LIN {X 0,Y 513.004,Z 916.305,A -85,B 0,C 180,E1 22393.038,E2 22393.038} C_VEL
LIN {X 0,Y 508.896,Z 933.803,A -85,B 0,C 180,E1 22391.855,E2 22391.855} C_VEL
LIN {X 0,Y 504.363,Z 951.797,A -85,B 0,C 180,E1 22390.486,E2 22390.486} C_VEL
LIN {X 0,Y 498.956,Z 972.158,A -85,B 0,C 180,E1 22388.725,E2 22388.725} C_VEL
LIN {X 0,Y 493.08,Z 992.756,A -85,B 0,C 180,E1 22386.651,E2 22386.651} C_VEL
LIN {X 0,Y 488.236,Z 1008.925,A -85,B 0,C 180,E1 22384.788,E2 22384.788} C_VEL
LIN {X 0,Y 483.886,Z 1023.135,A -85,B 0,C 180,E1 22382.95,E2 22382.95} C_VEL
LIN {X 0,Y 479.724,Z 1036.506,A -85,B 0,C 180,E1 22381.021,E2 22381.021} C_VEL
LIN {X 0,Y 475.565,Z 1049.952,A -85,B 0,C 180,E1 22378.841,E2 22378.841} C_VEL
LIN {X 0,Y 470.95,Z 1065.021,A -85,B 0,C 180,E1 22376.057,E2 22376.057} C_VEL
LIN {X 0,Y 466.983,Z 1078.097,A -85,B 0,C 180,E1 22373.207,E2 22373.207} C_VEL
LIN {X 0,Y 464.273,Z 1087.644,A -85,B 0,C 180,E1 22370.835,E2 22370.835} C_VEL
LIN {X 0,Y 461.919,Z 1096.543,A -85,B 0,C 180,E1 22368.315,E2 22368.315} C_VEL
LIN {X 0,Y 459.756,Z 1105.63,A -85,B 0,C 180,E1 22365.33,E2 22365.33} C_VEL
LIN {X 0,Y 457.961,Z 1114.229,A -85,B 0,C 180,E1 22361.883,E2 22361.883} C_VEL
LIN {X 0,Y 456.92,Z 1120.716,A -85,B 0,C 180,E1 22358.628,E2 22358.628} C_VEL
LIN {X 0,Y 456.305,Z 1125.981,A -85,B 0,C 180,E1 22355.181,E2 22355.181} C_VEL
LIN {X 0,Y 456.039,Z 1129.45,A -85,B 0,C 180,E1 22351.898,E2 22351.898} C_VEL
LIN {X 0,Y 455.95,Z 1131.611,A -85,B 0,C 180,E1 22348.696,E2 22348.696} C_VEL
LIN {X 0,Y 455.919,Z 1132.456,A -85,B 0,C 180,E1 22345.371,E2 22345.371} C_VEL
LIN {X 0,Y 455.939,Z 1131.95,A -85,B 0,C 180,E1 22342.025,E2 22342.025} C_VEL
LIN {X 0,Y 456.017,Z 1130.259,A -85,B 0,C 180,E1 22338.803,E2 22338.803} C_VEL
LIN {X 0,Y 456.242,Z 1127.297,A -85,B 0,C 180,E1 22335.638,E2 22335.638} C_VEL
LIN {X 0,Y 456.832,Z 1122.324,A -85,B 0,C 180,E1 22331.943,E2 22331.943} C_VEL
LIN {X 0,Y 457.747,Z 1116.901,A -85,B 0,C 180,E1 22328.922,E2 22328.922} C_VEL
LIN {X 0,Y 459.142,Z 1110.45,A -85,B 0,C 180,E1 22326,E2 22326} C_VEL
LIN {X 0,Y 461.433,Z 1101.534,A -85,B 0,C 180,E1 22322.646,E2 22322.646} C_VEL
LIN {X 0,Y 464.2,Z 1091.739,A -85,B 0,C 180,E1 22319.63,E2 22319.63} C_VEL
LIN {X 0,Y 467.056,Z 1082.545,A -85,B 0,C 180,E1 22317.178,E2 22317.178} C_VEL
LIN {X 0,Y 470.587,Z 1071.658,A -85,B 0,C 180,E1 22314.636,E2 22314.636} C_VEL
LIN {X 0,Y 475.522,Z 1056.822,A -85,B 0,C 180,E1 22311.658,E2 22311.658} C_VEL
LIN {X 0,Y 480.059,Z 1043.222,A -85,B 0,C 180,E1 22309.317,E2 22309.317} C_VEL
LIN {X 0,Y 484.312,Z 1030.344,A -85,B 0,C 180,E1 22307.359,E2 22307.359} C_VEL
LIN {X 0,Y 489.507,Z 1014.375,A -85,B 0,C 180,E1 22305.207,E2 22305.207} C_VEL
LIN {X 0,Y 495.258,Z 995.651,A -85,B 0,C 180,E1 22303.038,E2 22303.038} C_VEL
LIN {X 0,Y 500.116,Z 978.885,A -85,B 0,C 180,E1 22301.344,E2 22301.344} C_VEL
LIN {X 0,Y 504.892,Z 961.372,A -85,B 0,C 180,E1 22299.783,E2 22299.783} C_VEL
LIN {X 0,Y 510.558,Z 938.629,A -85,B 0,C 180,E1 22298.034,E2 22298.034} C_VEL
LIN {X 0,Y 514.787,Z 919.641,A -85,B 0,C 180,E1 22296.778,E2 22296.778} C_VEL
LIN {X 0,Y 518.75,Z 899.981,A -85,B 0,C 180,E1 22295.639,E2 22295.639} C_VEL
LIN {X 0,Y 523.349,Z 873.872,A -85,B 0,C 180,E1 22294.358,E2 22294.358} C_VEL
LIN {X 0,Y 526.811,Z 850.592,A -85,B 0,C 180,E1 22293.412,E2 22293.412} C_VEL
LIN {X 0,Y 530.26,Z 822.527,A -85,B 0,C 180,E1 22292.484,E2 22292.484} C_VEL
LIN {X 0,Y 532.541,Z 798.965,A -85,B 0,C 180,E1 22291.871,E2 22291.871} C_VEL
LIN {X 0,Y 537.311,Z 750.366,A -85,B 0,C 180,E1 22290.881,E2 22290.881} C_VEL
LIN {X 0,Y 544.533,Z 694.845,A -85,B 0,C 180,E1 22289.755,E2 22289.755} C_VEL
LIN {X 0,Y 553.51,Z 640.553,A -85,B 0,C 180,E1 22288.628,E2 22288.628} C_VEL
LIN {X 0,Y 556.071,Z 627.061,A -85,B 0,C 180,E1 22288.34,E2 22288.34} C_VEL
LIN {X 0,Y 546.521,Z 681.856,A -85,B 0,C 180,E1 22287.174,E2 22287.174} C_VEL
LIN {X 0,Y 538.863,Z 737.457,A -85,B 0,C 180,E1 22286.009,E2 22286.009} C_VEL
LIN {X 0,Y 532.662,Z 796.426,A -85,B 0,C 180,E1 22284.834,E2 22284.834} C_VEL
LIN {X 0,Y 526.114,Z 872.476,A -85,B 0,C 180,E1 22283.357,E2 22283.357} C_VEL
LIN {X 0,Y 522.106,Z 907.176,A -85,B 0,C 180,E1 22282.53,E2 22282.53} C_VEL
LIN {X 0,Y 517.848,Z 936.61,A -85,B 0,C 180,E1 22281.665,E2 22281.665} C_VEL
LIN {X 0,Y 514.037,Z 961.449,A -85,B 0,C 180,E1 22280.789,E2 22280.789} C_VEL
LIN {X 0,Y 509.447,Z 989.993,A -85,B 0,C 180,E1 22279.598,E2 22279.598} C_VEL
LIN {X 0,Y 504.721,Z 1017.061,A -85,B 0,C 180,E1 22278.242,E2 22278.242} C_VEL
LIN {X 0,Y 500.707,Z 1039.308,A -85,B 0,C 180,E1 22276.96,E2 22276.96} C_VEL
LIN {X 0,Y 496.772,Z 1060.139,A -85,B 0,C 180,E1 22275.604,E2 22275.604} C_VEL
LIN {X 0,Y 492.42,Z 1082.294,A -85,B 0,C 180,E1 22273.983,E2 22273.983} C_VEL
LIN {X 0,Y 487.088,Z 1108.576,A -85,B 0,C 180,E1 22271.762,E2 22271.762} C_VEL
LIN {X 0,Y 483.055,Z 1127.63,A -85,B 0,C 180,E1 22269.916,E2 22269.916} C_VEL
LIN {X 0,Y 479.373,Z 1144.946,A -85,B 0,C 180,E1 22268.05,E2 22268.05} C_VEL
LIN {X 0,Y 475.899,Z 1161.134,A -85,B 0,C 180,E1 22266.11,E2 22266.11} C_VEL
LIN {X 0,Y 472.666,Z 1176.256,A -85,B 0,C 180,E1 22264.096,E2 22264.096} C_VEL
LIN {X 0,Y 469.674,Z 1190.375,A -85,B 0,C 180,E1 22262.011,E2 22262.011} C_VEL
LIN {X 0,Y 466.886,Z 1203.851,A -85,B 0,C 180,E1 22259.792,E2 22259.792} C_VEL
LIN {X 0,Y 464.283,Z 1217.349,A -85,B 0,C 180,E1 22257.304,E2 22257.304} C_VEL
LIN {X 0,Y 461.559,Z 1232.06,A -85,B 0,C 180,E1 22254.169,E2 22254.169} C_VEL
LIN {X 0,Y 459.824,Z 1242.603,A -85,B 0,C 180,E1 22251.561,E2 22251.561} C_VEL
LIN {X 0,Y 458.528,Z 1251.331,A -85,B 0,C 180,E1 22249.092,E2 22249.092} C_VEL
LIN {X 0,Y 457.561,Z 1258.863,A -85,B 0,C 180,E1 22246.634,E2 22246.634} C_VEL
LIN {X 0,Y 456.827,Z 1265.33,A -85,B 0,C 180,E1 22244.156,E2 22244.156} C_VEL
LIN {X 0,Y 456.384,Z 1270.815,A -85,B 0,C 180,E1 22241.628,E2 22241.628} C_VEL
LIN {X 0,Y 456.074,Z 1275.217,A -85,B 0,C 180,E1 22239.082,E2 22239.082} C_VEL
LIN {X 0,Y 455.965,Z 1278.515,A -85,B 0,C 180,E1 22236.548,E2 22236.548} C_VEL
LIN {X 0,Y 455.919,Z 1280.569,A -85,B 0,C 180,E1 22234.15,E2 22234.15} C_VEL
LIN {X 0,Y 455.905,Z 1281.679,A -85,B 0,C 180,E1 22231.634,E2 22231.634} C_VEL
LIN {X 0,Y 455.869,Z 1281.819,A -85,B 0,C 180,E1 22229.12,E2 22229.12} C_VEL
LIN {X 0,Y 455.911,Z 1281.009,A -85,B 0,C 180,E1 22226.605,E2 22226.605} C_VEL
LIN {X 0,Y 455.946,Z 1279.161,A -85,B 0,C 180,E1 22224.084,E2 22224.084} C_VEL
LIN {X 0,Y 456.058,Z 1276,A -85,B 0,C 180,E1 22221.419,E2 22221.419} C_VEL
LIN {X 0,Y 456.296,Z 1271.935,A -85,B 0,C 180,E1 22218.882,E2 22218.882} C_VEL
LIN {X 0,Y 456.709,Z 1266.786,A -85,B 0,C 180,E1 22216.323,E2 22216.323} C_VEL
LIN {X 0,Y 457.378,Z 1260.539,A -85,B 0,C 180,E1 22213.75,E2 22213.75} C_VEL
LIN {X 0,Y 458.351,Z 1253.158,A -85,B 0,C 180,E1 22211.164,E2 22211.164} C_VEL
LIN {X 0,Y 459.767,Z 1244.151,A -85,B 0,C 180,E1 22208.437,E2 22208.437} C_VEL
LIN {X 0,Y 462.054,Z 1231.676,A -85,B 0,C 180,E1 22205.177,E2 22205.177} C_VEL
LIN {X 0,Y 464.711,Z 1218.784,A -85,B 0,C 180,E1 22202.306,E2 22202.306} C_VEL
LIN {X 0,Y 467.503,Z 1206.27,A -85,B 0,C 180,E1 22199.827,E2 22199.827} C_VEL
LIN {X 0,Y 470.696,Z 1193.091,A -85,B 0,C 180,E1 22197.491,E2 22197.491} C_VEL
LIN {X 0,Y 474.609,Z 1177.626,A -85,B 0,C 180,E1 22195.038,E2 22195.038} C_VEL
LIN {X 0,Y 479.833,Z 1157.318,A -85,B 0,C 180,E1 22192.22,E2 22192.22} C_VEL
LIN {X 0,Y 484.33,Z 1140.198,A -85,B 0,C 180,E1 22190.133,E2 22190.133} C_VEL
LIN {X 0,Y 488.847,Z 1123.039,A -85,B 0,C 180,E1 22188.259,E2 22188.259} C_VEL
LIN {X 0,Y 493.602,Z 1104.685,A -85,B 0,C 180,E1 22186.47,E2 22186.47} C_VEL
LIN {X 0,Y 499.885,Z 1079.832,A -85,B 0,C 180,E1 22184.361,E2 22184.361} C_VEL
LIN {X 0,Y 504.754,Z 1059.498,A -85,B 0,C 180,E1 22182.867,E2 22182.867} C_VEL
LIN {X 0,Y 509.301,Z 1039.584,A -85,B 0,C 180,E1 22181.574,E2 22181.574} C_VEL
LIN {X 0,Y 513.825,Z 1018.51,A -85,B 0,C 180,E1 22180.374,E2 22180.374} C_VEL
LIN {X 0,Y 519.014,Z 992.538,A -85,B 0,C 180,E1 22179.114,E2 22179.114} C_VEL
LIN {X 0,Y 523.352,Z 967.608,A -85,B 0,C 180,E1 22178.126,E2 22178.126} C_VEL
LIN {X 0,Y 526.751,Z 945.768,A -85,B 0,C 180,E1 22177.406,E2 22177.406} C_VEL
LIN {X 0,Y 529.722,Z 923.918,A -85,B 0,C 180,E1 22176.817,E2 22176.817} C_VEL
LIN {X 0,Y 532.706,Z 896.601,A -85,B 0,C 180,E1 22176.227,E2 22176.227} C_VEL
LIN {X 0,Y 535.346,Z 850.987,A -85,B 0,C 180,E1 22175.476,E2 22175.476} C_VEL
LIN {X 0,Y 546.358,Z 652.974,A -85,B 0,C 180,E1 22172.307,E2 22172.307} C_VEL
LIN {X 0,Y 555.509,Z 504.464,A -85,B 0,C 180,E1 22169.877,E2 22169.877} C_VEL
LIN {X 0,Y 542.54,Z 483.994,A -85,B 0,C 180,E1 22167.198,E2 22167.198} C_VEL
LIN {X 0,Y 530.395,Z 465.804,A -85,B 0,C 180,E1 22164.444,E2 22164.444} C_VEL
LIN {X 0,Y 519.173,Z 449.741,A -85,B 0,C 180,E1 22161.643,E2 22161.643} C_VEL
LIN {X 0,Y 511.694,Z 439.449,A -85,B 0,C 180,E1 22159.64,E2 22159.64} C_VEL
LIN {X 0,Y 505.445,Z 430.708,A -85,B 0,C 180,E1 22157.797,E2 22157.797} C_VEL
LIN {X 0,Y 500.388,Z 423.97,A -85,B 0,C 180,E1 22156.245,E2 22156.245} C_VEL
LIN {X 0,Y 493.447,Z 414.591,A -85,B 0,C 180,E1 22153.927,E2 22153.927} C_VEL
LIN {X 0,Y 488.699,Z 408.401,A -85,B 0,C 180,E1 22152.226,E2 22152.226} C_VEL
LIN {X 0,Y 485.165,Z 403.669,A -85,B 0,C 180,E1 22150.87,E2 22150.87} C_VEL
LIN {X 0,Y 480.579,Z 397.719,A -85,B 0,C 180,E1 22149.038,E2 22149.038} C_VEL
LIN {X 0,Y 476.464,Z 392.336,A -85,B 0,C 180,E1 22147.234,E2 22147.234} C_VEL
LIN {X 0,Y 473.078,Z 388.046,A -85,B 0,C 180,E1 22145.701,E2 22145.701} C_VEL
LIN {X 0,Y 471.648,Z 386.105,A -85,B 0,C 180,E1 22144.986,E2 22144.986} C_VEL
LIN {X 0,Y 469.016,Z 382.07,A -85,B 0,C 180,E1 22143.3,E2 22143.3} C_VEL
LIN {X 0,Y 467.992,Z 380.45,A -85,B 0,C 180,E1 22142.572,E2 22142.572} C_VEL
LIN {X 0,Y 465.751,Z 376.915,A -85,B 0,C 180,E1 22140.861,E2 22140.861} C_VEL
LIN {X 0,Y 464.943,Z 375.295,A -85,B 0,C 180,E1 22140.106,E2 22140.106} C_VEL
LIN {X 0,Y 462.408,Z 371.852,A -85,B 0,C 180,E1 22138.141,E2 22138.141} C_VEL
LIN {X 0,Y 461.444,Z 369.713,A -85,B 0,C 180,E1 22137.143,E2 22137.143} C_VEL
LIN {X 0,Y 458.88,Z 366.479,A -85,B 0,C 180,E1 22135,E2 22135} C_VEL
LIN {X 0,Y 458.244,Z 364.355,A -85,B 0,C 180,E1 22133.862,E2 22133.862} C_VEL
LIN {X 0,Y 458.239,Z 364.153,A -85,B 0,C 180,E1 22130.327,E2 22130.327} C_VEL
LIN {X 0,Y 458.227,Z 364.151,A -85,B 0,C 180,E1 22126.626,E2 22126.626} C_VEL
LIN {X 0,Y 458.199,Z 364.14,A -85,B 0,C 180,E1 22122.997,E2 22122.997} C_VEL
LIN {X 0,Y 458.203,Z 364.141,A -85,B 0,C 180,E1 22119.297,E2 22119.297} C_VEL
LIN {X 0,Y 458.237,Z 364.14,A -85,B 0,C 180,E1 22115.781,E2 22115.781} C_VEL
LIN {X 0,Y 458.235,Z 364.153,A -85,B 0,C 180,E1 22112.021,E2 22112.021} C_VEL
LIN {X 0,Y 458.199,Z 364.152,A -85,B 0,C 180,E1 22108.417,E2 22108.417} C_VEL
LIN {X 0,Y 458.191,Z 364.143,A -85,B 0,C 180,E1 22104.669,E2 22104.669} C_VEL
LIN {X 0,Y 458.215,Z 364.138,A -85,B 0,C 180,E1 22101.063,E2 22101.063} C_VEL
LIN {X 0,Y 458.23,Z 364.137,A -85,B 0,C 180,E1 22097.521,E2 22097.521} C_VEL
LIN {X 0,Y 458.191,Z 364.146,A -85,B 0,C 180,E1 22093.933,E2 22093.933} C_VEL
LIN {X 0,Y 458.185,Z 364.157,A -85,B 0,C 180,E1 22090.237,E2 22090.237} C_VEL
LIN {X 0,Y 458.215,Z 364.152,A -85,B 0,C 180,E1 22086.719,E2 22086.719} C_VEL
LIN {X 0,Y 458.223,Z 364.141,A -85,B 0,C 180,E1 22083.06,E2 22083.06} C_VEL
LIN {X 0,Y 458.179,Z 364.14,A -85,B 0,C 180,E1 22079.551,E2 22079.551} C_VEL
LIN {X 0,Y 458.177,Z 364.141,A -85,B 0,C 180,E1 22075.878,E2 22075.878} C_VEL
LIN {X 0,Y 458.239,Z 364.483,A -85,B 0,C 180,E1 22073.126,E2 22073.126} C_VEL
LIN {X 0,Y 458.73,Z 366.115,A -85,B 0,C 180,E1 22072.423,E2 22072.423} C_VEL
LIN {X 0,Y 460.215,Z 368.566,A -85,B 0,C 180,E1 22071.475,E2 22071.475} C_VEL
LIN {X 0,Y 464.25,Z 371.568,A -85,B 0,C 180,E1 22069.371,E2 22069.371} C_VEL
LIN {X 0,Y 466.378,Z 375.19,A -85,B 0,C 180,E1 22068.183,E2 22068.183} C_VEL
LIN {X 0,Y 469.791,Z 377.548,A -85,B 0,C 180,E1 22066.641,E2 22066.641} C_VEL
LIN {X 0,Y 472.178,Z 381.527,A -85,B 0,C 180,E1 22065.475,E2 22065.475} C_VEL
LIN {X 0,Y 475.855,Z 384.645,A -85,B 0,C 180,E1 22063.952,E2 22063.952} C_VEL
LIN {X 0,Y 478.445,Z 388.397,A -85,B 0,C 180,E1 22062.86,E2 22062.86} C_VEL
LIN {X 0,Y 481.486,Z 391.076,A -85,B 0,C 180,E1 22061.712,E2 22061.712} C_VEL
LIN {X 0,Y 484.417,Z 395.132,A -85,B 0,C 180,E1 22060.586,E2 22060.586} C_VEL
LIN {X 0,Y 487.024,Z 397.549,A -85,B 0,C 180,E1 22059.692,E2 22059.692} C_VEL
LIN {X 0,Y 490.367,Z 401.834,A -85,B 0,C 180,E1 22058.525,E2 22058.525} C_VEL
LIN {X 0,Y 492.345,Z 403.85,A -85,B 0,C 180,E1 22057.879,E2 22057.879} C_VEL
LIN {X 0,Y 495.969,Z 408.271,A -85,B 0,C 180,E1 22056.715,E2 22056.715} C_VEL
LIN {X 0,Y 497.697,Z 410.189,A -85,B 0,C 180,E1 22056.192,E2 22056.192} C_VEL
LIN {X 0,Y 501.825,Z 414.972,A -85,B 0,C 180,E1 22054.957,E2 22054.957} C_VEL
LIN {X 0,Y 508.371,Z 423.193,A -85,B 0,C 180,E1 22053.101,E2 22053.101} C_VEL
LIN {X 0,Y 512.691,Z 428.465,A -85,B 0,C 180,E1 22051.956,E2 22051.956} C_VEL
LIN {X 0,Y 520.517,Z 437.909,A -85,B 0,C 180,E1 22050,E2 22050} C_VEL
LIN {X 0,Y 533.39,Z 454.62,A -85,B 0,C 180,E1 22047.045,E2 22047.045} C_VEL
LIN {X 0,Y 546.906,Z 472.765,A -85,B 0,C 180,E1 22044.255,E2 22044.255} C_VEL
LIN {X 0,Y 551.745,Z 479.921,A -85,B 0,C 180,E1 22043.308,E2 22043.308} C_VEL
LIN {X 0,Y 541.721,Z 646.742,A -85,B 0,C 180,E1 22040.63,E2 22040.63} C_VEL
LIN {X 0,Y 540.695,Z 654.432,A -85,B 0,C 180,E1 22040.593,E2 22040.593} C_VEL
LIN {X 0,Y 535.758,Z 675.009,A -85,B 0,C 180,E1 22040.799,E2 22040.799} C_VEL
LIN {X 0,Y 534.919,Z 681.606,A -85,B 0,C 180,E1 22040.757,E2 22040.757} C_VEL
LIN {X 0,Y 529.459,Z 774.436,A -85,B 0,C 180,E1 22039.25,E2 22039.25} C_VEL
LIN {X 0,Y 526.721,Z 803.495,A -85,B 0,C 180,E1 22038.601,E2 22038.601} C_VEL
LIN {X 0,Y 523.864,Z 826.675,A -85,B 0,C 180,E1 22037.922,E2 22037.922} C_VEL
LIN {X 0,Y 520.738,Z 848.037,A -85,B 0,C 180,E1 22037.164,E2 22037.164} C_VEL
LIN {X 0,Y 516.555,Z 872.837,A -85,B 0,C 180,E1 22036.112,E2 22036.112} C_VEL
LIN {X 0,Y 511.514,Z 898.023,A -85,B 0,C 180,E1 22034.815,E2 22034.815} C_VEL
LIN {X 0,Y 507.372,Z 916.835,A -85,B 0,C 180,E1 22033.688,E2 22033.688} C_VEL
LIN {X 0,Y 503.076,Z 934.617,A -85,B 0,C 180,E1 22032.482,E2 22032.482} C_VEL
LIN {X 0,Y 498.376,Z 952.74,A -85,B 0,C 180,E1 22031.094,E2 22031.094} C_VEL
LIN {X 0,Y 492.752,Z 973.294,A -85,B 0,C 180,E1 22029.304,E2 22029.304} C_VEL
LIN {X 0,Y 486.729,Z 993.783,A -85,B 0,C 180,E1 22027.224,E2 22027.224} C_VEL
LIN {X 0,Y 481.743,Z 1010.033,A -85,B 0,C 180,E1 22025.343,E2 22025.343} C_VEL
LIN {X 0,Y 477.107,Z 1024.689,A -85,B 0,C 180,E1 22023.428,E2 22023.428} C_VEL
LIN {X 0,Y 472.642,Z 1038.539,A -85,B 0,C 180,E1 22021.396,E2 22021.396} C_VEL
LIN {X 0,Y 467.655,Z 1054.24,A -85,B 0,C 180,E1 22018.787,E2 22018.787} C_VEL
LIN {X 0,Y 462.991,Z 1068.633,A -85,B 0,C 180,E1 22015.99,E2 22015.99} C_VEL
LIN {X 0,Y 459.604,Z 1079.519,A -85,B 0,C 180,E1 22013.565,E2 22013.565} C_VEL
LIN {X 0,Y 456.82,Z 1088.918,A -85,B 0,C 180,E1 22011.189,E2 22011.189} C_VEL
LIN {X 0,Y 454.497,Z 1097.265,A -85,B 0,C 180,E1 22008.799,E2 22008.799} C_VEL
LIN {X 0,Y 452.489,Z 1105.073,A -85,B 0,C 180,E1 22006.24,E2 22006.24} C_VEL
LIN {X 0,Y 450.753,Z 1112.712,A -85,B 0,C 180,E1 22003.316,E2 22003.316} C_VEL
LIN {X 0,Y 449.347,Z 1120.434,A -85,B 0,C 180,E1 21999.654,E2 21999.654} C_VEL
LIN {X 0,Y 448.558,Z 1125.77,A -85,B 0,C 180,E1 21996.367,E2 21996.367} C_VEL
LIN {X 0,Y 448.2,Z 1129.589,A -85,B 0,C 180,E1 21993.22,E2 21993.22} C_VEL
LIN {X 0,Y 448.075,Z 1132.274,A -85,B 0,C 180,E1 21989.844,E2 21989.844} C_VEL
LIN {X 0,Y 448,Z 1133.571,A -85,B 0,C 180,E1 21986.655,E2 21986.655} C_VEL
LIN {X 0,Y 448.027,Z 1133.654,A -85,B 0,C 180,E1 21983.686,E2 21983.686} C_VEL
LIN {X 0,Y 448.09,Z 1132.642,A -85,B 0,C 180,E1 21980.372,E2 21980.372} C_VEL
LIN {X 0,Y 448.259,Z 1130.095,A -85,B 0,C 180,E1 21976.857,E2 21976.857} C_VEL
LIN {X 0,Y 448.595,Z 1126.653,A -85,B 0,C 180,E1 21973.798,E2 21973.798} C_VEL
LIN {X 0,Y 449.316,Z 1122.365,A -85,B 0,C 180,E1 21970.904,E2 21970.904} C_VEL
LIN {X 0,Y 450.442,Z 1116.579,A -85,B 0,C 180,E1 21967.782,E2 21967.782} C_VEL
LIN {X 0,Y 452.514,Z 1108.154,A -85,B 0,C 180,E1 21964.182,E2 21964.182} C_VEL
LIN {X 0,Y 454.751,Z 1100.236,A -85,B 0,C 180,E1 21961.386,E2 21961.386} C_VEL
LIN {X 0,Y 457.417,Z 1091.568,A -85,B 0,C 180,E1 21958.747,E2 21958.747} C_VEL
LIN {X 0,Y 461.372,Z 1079.746,A -85,B 0,C 180,E1 21955.65,E2 21955.65} C_VEL
LIN {X 0,Y 465.718,Z 1066.995,A -85,B 0,C 180,E1 21952.847,E2 21952.847} C_VEL
LIN {X 0,Y 469.852,Z 1055.188,A -85,B 0,C 180,E1 21950.569,E2 21950.569} C_VEL
LIN {X 0,Y 474.968,Z 1040.58,A -85,B 0,C 180,E1 21948.094,E2 21948.094} C_VEL
LIN {X 0,Y 480.911,Z 1023.013,A -85,B 0,C 180,E1 21945.552,E2 21945.552} C_VEL
LIN {X 0,Y 485.615,Z 1008.68,A -85,B 0,C 180,E1 21943.738,E2 21943.738} C_VEL
LIN {X 0,Y 490.799,Z 992.25,A -85,B 0,C 180,E1 21941.899,E2 21941.899} C_VEL
LIN {X 0,Y 497.288,Z 970.127,A -85,B 0,C 180,E1 21939.767,E2 21939.767} C_VEL
LIN {X 0,Y 502.348,Z 951.309,A -85,B 0,C 180,E1 21938.209,E2 21938.209} C_VEL
LIN {X 0,Y 507.993,Z 928.473,A -85,B 0,C 180,E1 21936.572,E2 21936.572} C_VEL
LIN {X 0,Y 512.635,Z 906.977,A -85,B 0,C 180,E1 21935.268,E2 21935.268} C_VEL
LIN {X 0,Y 516.484,Z 887.424,A -85,B 0,C 180,E1 21934.239,E2 21934.239} C_VEL
LIN {X 0,Y 520.79,Z 862.442,A -85,B 0,C 180,E1 21933.111,E2 21933.111} C_VEL
LIN {X 0,Y 524.411,Z 837.382,A -85,B 0,C 180,E1 21932.182,E2 21932.182} C_VEL
LIN {X 0,Y 527.867,Z 808.491,A -85,B 0,C 180,E1 21931.33,E2 21931.33} C_VEL
LIN {X 0,Y 532.114,Z 769.215,A -85,B 0,C 180,E1 21930.452,E2 21930.452} C_VEL
LIN {X 0,Y 539.873,Z 714.603,A -85,B 0,C 180,E1 21929.327,E2 21929.327} C_VEL
LIN {X 0,Y 548.257,Z 667.388,A -85,B 0,C 180,E1 21928.33,E2 21928.33} C_VEL
LIN {X 0,Y 538.687,Z 722.229,A -85,B 0,C 180,E1 21927.154,E2 21927.154} C_VEL
LIN {X 0,Y 531.446,Z 775.044,A -85,B 0,C 180,E1 21926.042,E2 21926.042} C_VEL
LIN {X 0,Y 525.162,Z 834.674,A -85,B 0,C 180,E1 21924.847,E2 21924.847} C_VEL
LIN {X 0,Y 521.302,Z 871.534,A -85,B 0,C 180,E1 21924.073,E2 21924.073} C_VEL
LIN {X 0,Y 516.828,Z 906.216,A -85,B 0,C 180,E1 21923.209,E2 21923.209} C_VEL
LIN {X 0,Y 512.267,Z 935.607,A -85,B 0,C 180,E1 21922.324,E2 21922.324} C_VEL
LIN {X 0,Y 507.281,Z 966.145,A -85,B 0,C 180,E1 21921.21,E2 21921.21} C_VEL
LIN {X 0,Y 502.079,Z 995.766,A -85,B 0,C 180,E1 21919.882,E2 21919.882} C_VEL
LIN {X 0,Y 497.876,Z 1018.781,A -85,B 0,C 180,E1 21918.685,E2 21918.685} C_VEL
LIN {X 0,Y 493.198,Z 1043.51,A -85,B 0,C 180,E1 21917.214,E2 21917.214} C_VEL
LIN {X 0,Y 487.768,Z 1070.775,A -85,B 0,C 180,E1 21915.321,E2 21915.321} C_VEL
LIN {X 0,Y 483.28,Z 1092.406,A -85,B 0,C 180,E1 21913.602,E2 21913.602} C_VEL
LIN {X 0,Y 478.883,Z 1112.905,A -85,B 0,C 180,E1 21911.763,E2 21911.763} C_VEL
LIN {X 0,Y 473.873,Z 1135.858,A -85,B 0,C 180,E1 21909.428,E2 21909.428} C_VEL
LIN {X 0,Y 469.277,Z 1156.403,A -85,B 0,C 180,E1 21907.007,E2 21907.007} C_VEL
LIN {X 0,Y 465.809,Z 1172.204,A -85,B 0,C 180,E1 21904.916,E2 21904.916} C_VEL
LIN {X 0,Y 462.642,Z 1186.696,A -85,B 0,C 180,E1 21902.782,E2 21902.782} C_VEL
LIN {X 0,Y 459.788,Z 1200.098,A -85,B 0,C 180,E1 21900.588,E2 21900.588} C_VEL
LIN {X 0,Y 457.238,Z 1212.462,A -85,B 0,C 180,E1 21898.329,E2 21898.329} C_VEL
LIN {X 0,Y 455.066,Z 1223.555,A -85,B 0,C 180,E1 21896.068,E2 21896.068} C_VEL
LIN {X 0,Y 453.21,Z 1233.869,A -85,B 0,C 180,E1 21893.71,E2 21893.71} C_VEL
LIN {X 0,Y 451.675,Z 1243.221,A -85,B 0,C 180,E1 21891.287,E2 21891.287} C_VEL
LIN {X 0,Y 450.514,Z 1250.969,A -85,B 0,C 180,E1 21889.005,E2 21889.005} C_VEL
LIN {X 0,Y 449.666,Z 1257.561,A -85,B 0,C 180,E1 21886.802,E2 21886.802} C_VEL
LIN {X 0,Y 448.952,Z 1263.67,A -85,B 0,C 180,E1 21884.444,E2 21884.444} C_VEL
LIN {X 0,Y 448.52,Z 1269.06,A -85,B 0,C 180,E1 21881.965,E2 21881.965} C_VEL
LIN {X 0,Y 448.178,Z 1273.573,A -85,B 0,C 180,E1 21879.373,E2 21879.373} C_VEL
LIN {X 0,Y 448.069,Z 1277.012,A -85,B 0,C 180,E1 21876.761,E2 21876.761} C_VEL
LIN {X 0,Y 448.015,Z 1279.287,A -85,B 0,C 180,E1 21874.224,E2 21874.224} C_VEL
LIN {X 0,Y 447.989,Z 1280.519,A -85,B 0,C 180,E1 21871.663,E2 21871.663} C_VEL
LIN {X 0,Y 447.947,Z 1280.712,A -85,B 0,C 180,E1 21869.233,E2 21869.233} C_VEL
LIN {X 0,Y 447.994,Z 1279.896,A -85,B 0,C 180,E1 21866.673,E2 21866.673} C_VEL
LIN {X 0,Y 448.032,Z 1277.899,A -85,B 0,C 180,E1 21863.979,E2 21863.979} C_VEL
LIN {X 0,Y 448.133,Z 1274.758,A -85,B 0,C 180,E1 21861.281,E2 21861.281} C_VEL
LIN {X 0,Y 448.37,Z 1270.67,A -85,B 0,C 180,E1 21858.683,E2 21858.683} C_VEL
LIN {X 0,Y 448.761,Z 1265.802,A -85,B 0,C 180,E1 21856.208,E2 21856.208} C_VEL
LIN {X 0,Y 449.442,Z 1259.598,A -85,B 0,C 180,E1 21853.588,E2 21853.588} C_VEL
LIN {X 0,Y 450.441,Z 1252.258,A -85,B 0,C 180,E1 21850.955,E2 21850.955} C_VEL
LIN {X 0,Y 451.82,Z 1243.745,A -85,B 0,C 180,E1 21848.311,E2 21848.311} C_VEL
LIN {X 0,Y 453.835,Z 1232.97,A -85,B 0,C 180,E1 21845.393,E2 21845.393} C_VEL
LIN {X 0,Y 456.89,Z 1218.675,A -85,B 0,C 180,E1 21842.074,E2 21842.074} C_VEL
LIN {X 0,Y 459.962,Z 1205.514,A -85,B 0,C 180,E1 21839.412,E2 21839.412} C_VEL
LIN {X 0,Y 463.258,Z 1192.411,A -85,B 0,C 180,E1 21837.05,E2 21837.05} C_VEL
LIN {X 0,Y 467.307,Z 1176.956,A -85,B 0,C 180,E1 21834.56,E2 21834.56} C_VEL
LIN {X 0,Y 472.79,Z 1156.582,A -85,B 0,C 180,E1 21831.686,E2 21831.686} C_VEL
LIN {X 0,Y 477.567,Z 1139.119,A -85,B 0,C 180,E1 21829.53,E2 21829.53} C_VEL
LIN {X 0,Y 482.253,Z 1121.873,A -85,B 0,C 180,E1 21827.636,E2 21827.636} C_VEL
LIN {X 0,Y 487.577,Z 1102.093,A -85,B 0,C 180,E1 21825.701,E2 21825.701} C_VEL
LIN {X 0,Y 493.885,Z 1077.802,A -85,B 0,C 180,E1 21823.642,E2 21823.642} C_VEL
LIN {X 0,Y 498.939,Z 1057.424,A -85,B 0,C 180,E1 21822.142,E2 21822.142} C_VEL
LIN {X 0,Y 503.414,Z 1038.437,A -85,B 0,C 180,E1 21820.909,E2 21820.909} C_VEL
LIN {X 0,Y 508.1,Z 1017.128,A -85,B 0,C 180,E1 21819.697,E2 21819.697} C_VEL
LIN {X 0,Y 513.626,Z 989.976,A -85,B 0,C 180,E1 21818.39,E2 21818.39} C_VEL
LIN {X 0,Y 517.844,Z 966.502,A -85,B 0,C 180,E1 21817.461,E2 21817.461} C_VEL
LIN {X 0,Y 521.295,Z 944.968,A -85,B 0,C 180,E1 21816.75,E2 21816.75} C_VEL
LIN {X 0,Y 524.325,Z 923.438,A -85,B 0,C 180,E1 21816.166,E2 21816.166} C_VEL
LIN {X 0,Y 527.308,Z 897.027,A -85,B 0,C 180,E1 21815.59,E2 21815.59} C_VEL
LIN {X 0,Y 529.766,Z 857.782,A -85,B 0,C 180,E1 21814.929,E2 21814.929} C_VEL
LIN {X 0,Y 541.808,Z 649.363,A -85,B 0,C 180,E1 21811.568,E2 21811.568} C_VEL
LIN {X 0,Y 550.806,Z 508.74,A -85,B 0,C 180,E1 21809.26,E2 21809.26} C_VEL
LIN {X 0,Y 538.711,Z 489.496,A -85,B 0,C 180,E1 21806.691,E2 21806.691} C_VEL
LIN {X 0,Y 526.982,Z 471.891,A -85,B 0,C 180,E1 21803.986,E2 21803.986} C_VEL
LIN {X 0,Y 516.436,Z 456.655,A -85,B 0,C 180,E1 21801.316,E2 21801.316} C_VEL
LIN {X 0,Y 508.78,Z 445.976,A -85,B 0,C 180,E1 21799.219,E2 21799.219} C_VEL
LIN {X 0,Y 502.692,Z 437.517,A -85,B 0,C 180,E1 21797.419,E2 21797.419} C_VEL
LIN {X 0,Y 497.583,Z 430.555,A -85,B 0,C 180,E1 21795.8,E2 21795.8} C_VEL
LIN {X 0,Y 490.895,Z 421.549,A -85,B 0,C 180,E1 21793.547,E2 21793.547} C_VEL
LIN {X 0,Y 486.038,Z 415.07,A -85,B 0,C 180,E1 21791.751,E2 21791.751} C_VEL
LIN {X 0,Y 482.902,Z 410.931,A -85,B 0,C 180,E1 21790.559,E2 21790.559} C_VEL
LIN {X 0,Y 478.399,Z 404.989,A -85,B 0,C 180,E1 21788.716,E2 21788.716} C_VEL
LIN {X 0,Y 474.392,Z 399.766,A -85,B 0,C 180,E1 21786.961,E2 21786.961} C_VEL
LIN {X 0,Y 470.959,Z 395.235,A -85,B 0,C 180,E1 21785.36,E2 21785.36} C_VEL
LIN {X 0,Y 469.277,Z 393.17,A -85,B 0,C 180,E1 21784.522,E2 21784.522} C_VEL
LIN {X 0,Y 465.996,Z 388.646,A -85,B 0,C 180,E1 21782.829,E2 21782.829} C_VEL
LIN {X 0,Y 462.35,Z 384.266,A -85,B 0,C 180,E1 21780.805,E2 21780.805} C_VEL
LIN {X 0,Y 460.943,Z 382.143,A -85,B 0,C 180,E1 21779.921,E2 21779.921} C_VEL
LIN {X 0,Y 457.989,Z 378.223,A -85,B 0,C 180,E1 21777.873,E2 21777.873} C_VEL
LIN {X 0,Y 457.115,Z 376.389,A -85,B 0,C 180,E1 21776.991,E2 21776.991} C_VEL
LIN {X 0,Y 454.591,Z 373.09,A -85,B 0,C 180,E1 21774.826,E2 21774.826} C_VEL
LIN {X 0,Y 453.509,Z 370.705,A -85,B 0,C 180,E1 21773.544,E2 21773.544} C_VEL
LIN {X 0,Y 450.75,Z 367.004,A -85,B 0,C 180,E1 21770.794,E2 21770.794} C_VEL
LIN {X 0,Y 450.295,Z 365.316,A -85,B 0,C 180,E1 21769.633,E2 21769.633} C_VEL
LIN {X 0,Y 450.304,Z 365.138,A -85,B 0,C 180,E1 21765.993,E2 21765.993} C_VEL
LIN {X 0,Y 450.296,Z 365.126,A -85,B 0,C 180,E1 21762.286,E2 21762.286} C_VEL
LIN {X 0,Y 450.27,Z 365.137,A -85,B 0,C 180,E1 21758.642,E2 21758.642} C_VEL
LIN {X 0,Y 450.26,Z 365.145,A -85,B 0,C 180,E1 21754.903,E2 21754.903} C_VEL
LIN {X 0,Y 450.269,Z 365.132,A -85,B 0,C 180,E1 21751.191,E2 21751.191} C_VEL
LIN {X 0,Y 450.296,Z 365.125,A -85,B 0,C 180,E1 21747.542,E2 21747.542} C_VEL
LIN {X 0,Y 450.285,Z 365.126,A -85,B 0,C 180,E1 21743.795,E2 21743.795} C_VEL
LIN {X 0,Y 450.253,Z 365.134,A -85,B 0,C 180,E1 21740.207,E2 21740.207} C_VEL
LIN {X 0,Y 450.252,Z 365.145,A -85,B 0,C 180,E1 21736.494,E2 21736.494} C_VEL
LIN {X 0,Y 450.27,Z 365.139,A -85,B 0,C 180,E1 21732.805,E2 21732.805} C_VEL
LIN {X 0,Y 450.299,Z 365.128,A -85,B 0,C 180,E1 21729.199,E2 21729.199} C_VEL
LIN {X 0,Y 450.252,Z 365.129,A -85,B 0,C 180,E1 21725.579,E2 21725.579} C_VEL
LIN {X 0,Y 450.24,Z 365.131,A -85,B 0,C 180,E1 21721.907,E2 21721.907} C_VEL
LIN {X 0,Y 450.269,Z 365.166,A -85,B 0,C 180,E1 21718.373,E2 21718.373} C_VEL
LIN {X 0,Y 450.423,Z 366.036,A -85,B 0,C 180,E1 21717.212,E2 21717.212} C_VEL
LIN {X 0,Y 452.367,Z 369.645,A -85,B 0,C 180,E1 21715.532,E2 21715.532} C_VEL
LIN {X 0,Y 456.364,Z 372.5,A -85,B 0,C 180,E1 21713.041,E2 21713.041} C_VEL
LIN {X 0,Y 458.197,Z 375.89,A -85,B 0,C 180,E1 21711.843,E2 21711.843} C_VEL
LIN {X 0,Y 462.348,Z 379.152,A -85,B 0,C 180,E1 21709.618,E2 21709.618} C_VEL
LIN {X 0,Y 464.745,Z 382.984,A -85,B 0,C 180,E1 21708.307,E2 21708.307} C_VEL
LIN {X 0,Y 468.089,Z 385.564,A -85,B 0,C 180,E1 21706.76,E2 21706.76} C_VEL
LIN {X 0,Y 470.518,Z 389.328,A -85,B 0,C 180,E1 21705.6,E2 21705.6} C_VEL
LIN {X 0,Y 473.845,Z 392.199,A -85,B 0,C 180,E1 21704.2,E2 21704.2} C_VEL
LIN {X 0,Y 476.863,Z 396.331,A -85,B 0,C 180,E1 21702.928,E2 21702.928} C_VEL
LIN {X 0,Y 479.469,Z 398.663,A -85,B 0,C 180,E1 21701.946,E2 21701.946} C_VEL
LIN {X 0,Y 482.751,Z 402.983,A -85,B 0,C 180,E1 21700.683,E2 21700.683} C_VEL
LIN {X 0,Y 484.866,Z 405.01,A -85,B 0,C 180,E1 21699.945,E2 21699.945} C_VEL
LIN {X 0,Y 488.535,Z 409.539,A -85,B 0,C 180,E1 21698.672,E2 21698.672} C_VEL
LIN {X 0,Y 490.191,Z 411.328,A -85,B 0,C 180,E1 21698.123,E2 21698.123} C_VEL
LIN {X 0,Y 494.098,Z 415.979,A -85,B 0,C 180,E1 21696.857,E2 21696.857} C_VEL
LIN {X 0,Y 500.741,Z 424.012,A -85,B 0,C 180,E1 21694.849,E2 21694.849} C_VEL
LIN {X 0,Y 505.541,Z 429.911,A -85,B 0,C 180,E1 21693.484,E2 21693.484} C_VEL
LIN {X 0,Y 514.56,Z 440.928,A -85,B 0,C 180,E1 21691.113,E2 21691.113} C_VEL
LIN {X 0,Y 522.502,Z 451.146,A -85,B 0,C 180,E1 21689.178,E2 21689.178} C_VEL
LIN {X 0,Y 531.353,Z 462.656,A -85,B 0,C 180,E1 21687.169,E2 21687.169} C_VEL
LIN {X 0,Y 544.3,Z 480.226,A -85,B 0,C 180,E1 21684.475,E2 21684.475} C_VEL
LIN {X 0,Y 546.995,Z 484.344,A -85,B 0,C 180,E1 21683.933,E2 21683.933} C_VEL
LIN {X 0,Y 534.919,Z 681.606,A -85,B 0,C 180,E1 21680.757,E2 21680.757} C_VEL
LIN {X 0,Y 533.863,Z 689.291,A -85,B 0,C 180,E1 21680.719,E2 21680.719} C_VEL
LIN {X 0,Y 528.839,Z 709.849,A -85,B 0,C 180,E1 21680.922,E2 21680.922} C_VEL
LIN {X 0,Y 527.983,Z 716.444,A -85,B 0,C 180,E1 21680.882,E2 21680.882} C_VEL
LIN {X 0,Y 524.23,Z 776.923,A -85,B 0,C 180,E1 21679.884,E2 21679.884} C_VEL
LIN {X 0,Y 521.436,Z 805.134,A -85,B 0,C 180,E1 21679.238,E2 21679.238} C_VEL
LIN {X 0,Y 518.544,Z 827.892,A -85,B 0,C 180,E1 21678.566,E2 21678.566} C_VEL
LIN {X 0,Y 515.274,Z 849.569,A -85,B 0,C 180,E1 21677.789,E2 21677.789} C_VEL
LIN {X 0,Y 510.714,Z 875.632,A -85,B 0,C 180,E1 21676.667,E2 21676.667} C_VEL
LIN {X 0,Y 505.802,Z 899.36,A -85,B 0,C 180,E1 21675.428,E2 21675.428} C_VEL
LIN {X 0,Y 501.443,Z 918.589,A -85,B 0,C 180,E1 21674.265,E2 21674.265} C_VEL
LIN {X 0,Y 497.012,Z 936.507,A -85,B 0,C 180,E1 21673.04,E2 21673.04} C_VEL
LIN {X 0,Y 491.995,Z 955.387,A -85,B 0,C 180,E1 21671.578,E2 21671.578} C_VEL
LIN {X 0,Y 485.395,Z 978.483,A -85,B 0,C 180,E1 21669.501,E2 21669.501} C_VEL
LIN {X 0,Y 479.986,Z 996.166,A -85,B 0,C 180,E1 21667.658,E2 21667.658} C_VEL
LIN {X 0,Y 475.068,Z 1011.678,A -85,B 0,C 180,E1 21665.835,E2 21665.835} C_VEL
LIN {X 0,Y 470.149,Z 1026.831,A -85,B 0,C 180,E1 21663.831,E2 21663.831} C_VEL
LIN {X 0,Y 464.982,Z 1042.477,A -85,B 0,C 180,E1 21661.486,E2 21661.486} C_VEL
LIN {X 0,Y 459.532,Z 1058.651,A -85,B 0,C 180,E1 21658.666,E2 21658.666} C_VEL
LIN {X 0,Y 455.565,Z 1070.611,A -85,B 0,C 180,E1 21656.27,E2 21656.27} C_VEL
LIN {X 0,Y 452.108,Z 1081.368,A -85,B 0,C 180,E1 21653.828,E2 21653.828} C_VEL
LIN {X 0,Y 449.077,Z 1091.259,A -85,B 0,C 180,E1 21651.27,E2 21651.27} C_VEL
LIN {X 0,Y 446.217,Z 1101.341,A -85,B 0,C 180,E1 21648.262,E2 21648.262} C_VEL
LIN {X 0,Y 443.723,Z 1110.999,A -85,B 0,C 180,E1 21644.78,E2 21644.78} C_VEL
LIN {X 0,Y 442.259,Z 1117.539,A -85,B 0,C 180,E1 21641.943,E2 21641.943} C_VEL
LIN {X 0,Y 441.345,Z 1122.789,A -85,B 0,C 180,E1 21639.205,E2 21639.205} C_VEL
LIN {X 0,Y 440.642,Z 1127.561,A -85,B 0,C 180,E1 21636.118,E2 21636.118} C_VEL
LIN {X 0,Y 440.276,Z 1131.562,A -85,B 0,C 180,E1 21632.564,E2 21632.564} C_VEL
LIN {X 0,Y 440.166,Z 1133.815,A -85,B 0,C 180,E1 21629.385,E2 21629.385} C_VEL
LIN {X 0,Y 440.132,Z 1134.925,A -85,B 0,C 180,E1 21626.151,E2 21626.151} C_VEL
LIN {X 0,Y 440.104,Z 1134.894,A -85,B 0,C 180,E1 21623.003,E2 21623.003} C_VEL
LIN {X 0,Y 440.241,Z 1133.628,A -85,B 0,C 180,E1 21619.642,E2 21619.642} C_VEL
LIN {X 0,Y 440.443,Z 1131.077,A -85,B 0,C 180,E1 21616.35,E2 21616.35} C_VEL
LIN {X 0,Y 440.797,Z 1127.913,A -85,B 0,C 180,E1 21613.512,E2 21613.512} C_VEL
LIN {X 0,Y 441.548,Z 1123.824,A -85,B 0,C 180,E1 21610.701,E2 21610.701} C_VEL
LIN {X 0,Y 442.628,Z 1118.594,A -85,B 0,C 180,E1 21607.79,E2 21607.79} C_VEL
LIN {X 0,Y 444.699,Z 1110.724,A -85,B 0,C 180,E1 21604.255,E2 21604.255} C_VEL
LIN {X 0,Y 447.211,Z 1102.185,A -85,B 0,C 180,E1 21601.153,E2 21601.153} C_VEL
LIN {X 0,Y 449.987,Z 1093.59,A -85,B 0,C 180,E1 21598.472,E2 21598.472} C_VEL
LIN {X 0,Y 453.923,Z 1082.38,A -85,B 0,C 180,E1 21595.452,E2 21595.452} C_VEL
LIN {X 0,Y 458.624,Z 1069.255,A -85,B 0,C 180,E1 21592.483,E2 21592.483} C_VEL
LIN {X 0,Y 462.903,Z 1057.517,A -85,B 0,C 180,E1 21590.175,E2 21590.175} C_VEL
LIN {X 0,Y 467.403,Z 1045.172,A -85,B 0,C 180,E1 21588.024,E2 21588.024} C_VEL
LIN {X 0,Y 473.512,Z 1028.22,A -85,B 0,C 180,E1 21585.446,E2 21585.446} C_VEL
LIN {X 0,Y 479.41,Z 1010.875,A -85,B 0,C 180,E1 21583.197,E2 21583.197} C_VEL
LIN {X 0,Y 484.909,Z 994.125,A -85,B 0,C 180,E1 21581.298,E2 21581.298} C_VEL
LIN {X 0,Y 491.46,Z 972.712,A -85,B 0,C 180,E1 21579.205,E2 21579.205} C_VEL
LIN {X 0,Y 496.885,Z 953.409,A -85,B 0,C 180,E1 21577.584,E2 21577.584} C_VEL
LIN {X 0,Y 502.744,Z 930.772,A -85,B 0,C 180,E1 21575.938,E2 21575.938} C_VEL
LIN {X 0,Y 507.584,Z 909.583,A -85,B 0,C 180,E1 21574.63,E2 21574.63} C_VEL
LIN {X 0,Y 512.029,Z 888.449,A -85,B 0,C 180,E1 21573.499,E2 21573.499} C_VEL
LIN {X 0,Y 516.739,Z 862.662,A -85,B 0,C 180,E1 21572.328,E2 21572.328} C_VEL
LIN {X 0,Y 520.747,Z 837.724,A -85,B 0,C 180,E1 21571.391,E2 21571.391} C_VEL
LIN {X 0,Y 524.399,Z 810.487,A -85,B 0,C 180,E1 21570.571,E2 21570.571} C_VEL
LIN {X 0,Y 529.334,Z 772.315,A -85,B 0,C 180,E1 21569.683,E2 21569.683} C_VEL
LIN {X 0,Y 538.281,Z 718.853,A -85,B 0,C 180,E1 21568.558,E2 21568.558} C_VEL
LIN {X 0,Y 540.376,Z 707.959,A -85,B 0,C 180,E1 21568.32,E2 21568.32} C_VEL
LIN {X 0,Y 531.325,Z 759.359,A -85,B 0,C 180,E1 21567.21,E2 21567.21} C_VEL
LIN {X 0,Y 524.034,Z 811.907,A -85,B 0,C 180,E1 21566.098,E2 21566.098} C_VEL
LIN {X 0,Y 517.602,Z 865.294,A -85,B 0,C 180,E1 21564.955,E2 21564.955} C_VEL
LIN {X 0,Y 512.505,Z 901.187,A -85,B 0,C 180,E1 21564.04,E2 21564.04} C_VEL
LIN {X 0,Y 507.193,Z 932.895,A -85,B 0,C 180,E1 21563.073,E2 21563.073} C_VEL
LIN {X 0,Y 501.628,Z 964.734,A -85,B 0,C 180,E1 21561.887,E2 21561.887} C_VEL
LIN {X 0,Y 496.421,Z 992.737,A -85,B 0,C 180,E1 21560.619,E2 21560.619} C_VEL
LIN {X 0,Y 491.711,Z 1017.304,A -85,B 0,C 180,E1 21559.33,E2 21559.33} C_VEL
LIN {X 0,Y 486.314,Z 1044.689,A -85,B 0,C 180,E1 21557.672,E2 21557.672} C_VEL
LIN {X 0,Y 480.97,Z 1070.154,A -85,B 0,C 180,E1 21555.858,E2 21555.858} C_VEL
LIN {X 0,Y 476.771,Z 1089.596,A -85,B 0,C 180,E1 21554.296,E2 21554.296} C_VEL
LIN {X 0,Y 472.308,Z 1109.833,A -85,B 0,C 180,E1 21552.479,E2 21552.479} C_VEL
LIN {X 0,Y 467.105,Z 1132.997,A -85,B 0,C 180,E1 21550.114,E2 21550.114} C_VEL
LIN {X 0,Y 462.284,Z 1153.741,A -85,B 0,C 180,E1 21547.661,E2 21547.661} C_VEL
LIN {X 0,Y 458.616,Z 1169.816,A -85,B 0,C 180,E1 21545.525,E2 21545.525} C_VEL
LIN {X 0,Y 455.432,Z 1183.916,A -85,B 0,C 180,E1 21543.439,E2 21543.439} C_VEL
LIN {X 0,Y 452.491,Z 1197.405,A -85,B 0,C 180,E1 21541.221,E2 21541.221} C_VEL
LIN {X 0,Y 449.876,Z 1209.651,A -85,B 0,C 180,E1 21538.981,E2 21538.981} C_VEL
LIN {X 0,Y 447.543,Z 1221.007,A -85,B 0,C 180,E1 21536.661,E2 21536.661} C_VEL
LIN {X 0,Y 445.662,Z 1231.043,A -85,B 0,C 180,E1 21534.369,E2 21534.369} C_VEL
LIN {X 0,Y 444.017,Z 1240.616,A -85,B 0,C 180,E1 21531.906,E2 21531.906} C_VEL
LIN {X 0,Y 442.751,Z 1248.729,A -85,B 0,C 180,E1 21529.526,E2 21529.526} C_VEL
LIN {X 0,Y 441.807,Z 1255.916,A -85,B 0,C 180,E1 21527.11,E2 21527.11} C_VEL
LIN {X 0,Y 441.078,Z 1262.086,A -85,B 0,C 180,E1 21524.708,E2 21524.708} C_VEL
LIN {X 0,Y 440.629,Z 1267.544,A -85,B 0,C 180,E1 21522.183,E2 21522.183} C_VEL
LIN {X 0,Y 440.295,Z 1271.93,A -85,B 0,C 180,E1 21519.674,E2 21519.674} C_VEL
LIN {X 0,Y 440.176,Z 1275.555,A -85,B 0,C 180,E1 21516.936,E2 21516.936} C_VEL
LIN {X 0,Y 440.124,Z 1277.847,A -85,B 0,C 180,E1 21514.43,E2 21514.43} C_VEL
LIN {X 0,Y 440.101,Z 1279.168,A -85,B 0,C 180,E1 21511.823,E2 21511.823} C_VEL
LIN {X 0,Y 440.052,Z 1279.417,A -85,B 0,C 180,E1 21509.219,E2 21509.219} C_VEL
LIN {X 0,Y 440.091,Z 1278.62,A -85,B 0,C 180,E1 21506.613,E2 21506.613} C_VEL
LIN {X 0,Y 440.115,Z 1276.762,A -85,B 0,C 180,E1 21504.001,E2 21504.001} C_VEL
LIN {X 0,Y 440.2,Z 1273.667,A -85,B 0,C 180,E1 21501.246,E2 21501.246} C_VEL
LIN {X 0,Y 440.429,Z 1269.64,A -85,B 0,C 180,E1 21498.609,E2 21498.609} C_VEL
LIN {X 0,Y 440.814,Z 1264.818,A -85,B 0,C 180,E1 21496.088,E2 21496.088} C_VEL
LIN {X 0,Y 441.468,Z 1259,A -85,B 0,C 180,E1 21493.554,E2 21493.554} C_VEL
LIN {X 0,Y 442.491,Z 1251.633,A -85,B 0,C 180,E1 21490.831,E2 21490.831} C_VEL
LIN {X 0,Y 443.876,Z 1243.339,A -85,B 0,C 180,E1 21488.181,E2 21488.181} C_VEL
LIN {X 0,Y 445.722,Z 1233.678,A -85,B 0,C 180,E1 21485.48,E2 21485.48} C_VEL
LIN {X 0,Y 448.378,Z 1221.57,A -85,B 0,C 180,E1 21482.509,E2 21482.509} C_VEL
LIN {X 0,Y 452.05,Z 1206.239,A -85,B 0,C 180,E1 21479.273,E2 21479.273} C_VEL
LIN {X 0,Y 455.636,Z 1192.471,A -85,B 0,C 180,E1 21476.728,E2 21476.728} C_VEL
LIN {X 0,Y 459.345,Z 1178.817,A -85,B 0,C 180,E1 21474.466,E2 21474.466} C_VEL
LIN {X 0,Y 463.928,Z 1162.366,A -85,B 0,C 180,E1 21472.025,E2 21472.025} C_VEL
LIN {X 0,Y 470.099,Z 1140.572,A -85,B 0,C 180,E1 21469.219,E2 21469.219} C_VEL
LIN {X 0,Y 474.926,Z 1123.45,A -85,B 0,C 180,E1 21467.288,E2 21467.288} C_VEL
LIN {X 0,Y 479.906,Z 1105.558,A -85,B 0,C 180,E1 21465.485,E2 21465.485} C_VEL
LIN {X 0,Y 485.265,Z 1085.941,A -85,B 0,C 180,E1 21463.73,E2 21463.73} C_VEL
LIN {X 0,Y 491.923,Z 1060.397,A -85,B 0,C 180,E1 21461.759,E2 21461.759} C_VEL
LIN {X 0,Y 497.152,Z 1038.908,A -85,B 0,C 180,E1 21460.337,E2 21460.337} C_VEL
LIN {X 0,Y 501.727,Z 1018.842,A -85,B 0,C 180,E1 21459.175,E2 21459.175} C_VEL
LIN {X 0,Y 506.316,Z 997.391,A -85,B 0,C 180,E1 21458.098,E2 21458.098} C_VEL
LIN {X 0,Y 511.652,Z 969.793,A -85,B 0,C 180,E1 21456.939,E2 21456.939} C_VEL
LIN {X 0,Y 515.702,Z 945.564,A -85,B 0,C 180,E1 21456.121,E2 21456.121} C_VEL
LIN {X 0,Y 518.873,Z 923.878,A -85,B 0,C 180,E1 21455.525,E2 21455.525} C_VEL
LIN {X 0,Y 521.686,Z 900.165,A -85,B 0,C 180,E1 21454.998,E2 21454.998} C_VEL
LIN {X 0,Y 524.354,Z 862.873,A -85,B 0,C 180,E1 21454.34,E2 21454.34} C_VEL
LIN {X 0,Y 536.261,Z 661.958,A -85,B 0,C 180,E1 21451.086,E2 21451.086} C_VEL
LIN {X 0,Y 546.157,Z 513.027,A -85,B 0,C 180,E1 21448.634,E2 21448.634} C_VEL
LIN {X 0,Y 535.057,Z 495.339,A -85,B 0,C 180,E1 21446.229,E2 21446.229} C_VEL
LIN {X 0,Y 523.907,Z 478.395,A -85,B 0,C 180,E1 21443.598,E2 21443.598} C_VEL
LIN {X 0,Y 513.583,Z 463.426,A -85,B 0,C 180,E1 21440.962,E2 21440.962} C_VEL
LIN {X 0,Y 503.849,Z 449.474,A -85,B 0,C 180,E1 21438.184,E2 21438.184} C_VEL
LIN {X 0,Y 495.7,Z 438.371,A -85,B 0,C 180,E1 21435.652,E2 21435.652} C_VEL
LIN {X 0,Y 488.615,Z 428.794,A -85,B 0,C 180,E1 21433.25,E2 21433.25} C_VEL
LIN {X 0,Y 483.711,Z 422.198,A -85,B 0,C 180,E1 21431.416,E2 21431.416} C_VEL
LIN {X 0,Y 480.653,Z 418.187,A -85,B 0,C 180,E1 21430.245,E2 21430.245} C_VEL
LIN {X 0,Y 476.371,Z 412.41,A -85,B 0,C 180,E1 21428.449,E2 21428.449} C_VEL
LIN {X 0,Y 472.331,Z 407.19,A -85,B 0,C 180,E1 21426.686,E2 21426.686} C_VEL
LIN {X 0,Y 468.912,Z 402.528,A -85,B 0,C 180,E1 21425.046,E2 21425.046} C_VEL
LIN {X 0,Y 464.383,Z 396.696,A -85,B 0,C 180,E1 21422.749,E2 21422.749} C_VEL
LIN {X 0,Y 460.342,Z 391.46,A -85,B 0,C 180,E1 21420.436,E2 21420.436} C_VEL
LIN {X 0,Y 459.208,Z 389.836,A -85,B 0,C 180,E1 21419.75,E2 21419.75} C_VEL
LIN {X 0,Y 455.717,Z 385.479,A -85,B 0,C 180,E1 21417.548,E2 21417.548} C_VEL
LIN {X 0,Y 454.539,Z 383.776,A -85,B 0,C 180,E1 21416.721,E2 21416.721} C_VEL
LIN {X 0,Y 451.491,Z 380.144,A -85,B 0,C 180,E1 21414.535,E2 21414.535} C_VEL
LIN {X 0,Y 450.219,Z 377.99,A -85,B 0,C 180,E1 21413.496,E2 21413.496} C_VEL
LIN {X 0,Y 447.077,Z 374.313,A -85,B 0,C 180,E1 21410.863,E2 21410.863} C_VEL
LIN {X 0,Y 445.829,Z 371.929,A -85,B 0,C 180,E1 21409.533,E2 21409.533} C_VEL
LIN {X 0,Y 442.948,Z 368.287,A -85,B 0,C 180,E1 21406.289,E2 21406.289} C_VEL
LIN {X 0,Y 442.361,Z 366.289,A -85,B 0,C 180,E1 21404.665,E2 21404.665} C_VEL
LIN {X 0,Y 442.323,Z 366.131,A -85,B 0,C 180,E1 21401.003,E2 21401.003} C_VEL
LIN {X 0,Y 442.326,Z 366.119,A -85,B 0,C 180,E1 21397.26,E2 21397.26} C_VEL
LIN {X 0,Y 442.347,Z 366.114,A -85,B 0,C 180,E1 21393.523,E2 21393.523} C_VEL
LIN {X 0,Y 442.364,Z 366.113,A -85,B 0,C 180,E1 21389.881,E2 21389.881} C_VEL
LIN {X 0,Y 442.325,Z 366.125,A -85,B 0,C 180,E1 21386.214,E2 21386.214} C_VEL
LIN {X 0,Y 442.313,Z 366.137,A -85,B 0,C 180,E1 21382.51,E2 21382.51} C_VEL
LIN {X 0,Y 442.326,Z 366.124,A -85,B 0,C 180,E1 21378.829,E2 21378.829} C_VEL
LIN {X 0,Y 442.35,Z 366.115,A -85,B 0,C 180,E1 21375.15,E2 21375.15} C_VEL
LIN {X 0,Y 442.349,Z 366.113,A -85,B 0,C 180,E1 21371.37,E2 21371.37} C_VEL
LIN {X 0,Y 442.309,Z 366.122,A -85,B 0,C 180,E1 21367.779,E2 21367.779} C_VEL
LIN {X 0,Y 442.316,Z 366.227,A -85,B 0,C 180,E1 21363.981,E2 21363.981} C_VEL
LIN {X 0,Y 442.58,Z 367.28,A -85,B 0,C 180,E1 21362.757,E2 21362.757} C_VEL
LIN {X 0,Y 444.21,Z 370.334,A -85,B 0,C 180,E1 21360.95,E2 21360.95} C_VEL
LIN {X 0,Y 448.546,Z 373.563,A -85,B 0,C 180,E1 21357.474,E2 21357.474} C_VEL
LIN {X 0,Y 450.649,Z 377.305,A -85,B 0,C 180,E1 21355.733,E2 21355.733} C_VEL
LIN {X 0,Y 454.664,Z 380.268,A -85,B 0,C 180,E1 21353.213,E2 21353.213} C_VEL
LIN {X 0,Y 456.383,Z 383.48,A -85,B 0,C 180,E1 21352.065,E2 21352.065} C_VEL
LIN {X 0,Y 460.002,Z 386.235,A -85,B 0,C 180,E1 21350.111,E2 21350.111} C_VEL
LIN {X 0,Y 461.057,Z 387.928,A -85,B 0,C 180,E1 21349.51,E2 21349.51} C_VEL
LIN {X 0,Y 463.806,Z 391.444,A -85,B 0,C 180,E1 21348.086,E2 21348.086} C_VEL
LIN {X 0,Y 466.236,Z 393.343,A -85,B 0,C 180,E1 21346.957,E2 21346.957} C_VEL
LIN {X 0,Y 468.839,Z 397.136,A -85,B 0,C 180,E1 21345.715,E2 21345.715} C_VEL
LIN {X 0,Y 471.864,Z 399.759,A -85,B 0,C 180,E1 21344.442,E2 21344.442} C_VEL
LIN {X 0,Y 475.094,Z 404.063,A -85,B 0,C 180,E1 21343.07,E2 21343.07} C_VEL
LIN {X 0,Y 477.492,Z 406.284,A -85,B 0,C 180,E1 21342.168,E2 21342.168} C_VEL
LIN {X 0,Y 480.909,Z 410.656,A -85,B 0,C 180,E1 21340.846,E2 21340.846} C_VEL
LIN {X 0,Y 482.805,Z 412.59,A -85,B 0,C 180,E1 21340.169,E2 21340.169} C_VEL
LIN {X 0,Y 486.705,Z 417.243,A -85,B 0,C 180,E1 21338.82,E2 21338.82} C_VEL
LIN {X 0,Y 488.824,Z 419.924,A -85,B 0,C 180,E1 21338.098,E2 21338.098} C_VEL
LIN {X 0,Y 493.28,Z 425.138,A -85,B 0,C 180,E1 21336.662,E2 21336.662} C_VEL
LIN {X 0,Y 498.844,Z 431.861,A -85,B 0,C 180,E1 21334.996,E2 21334.996} C_VEL
LIN {X 0,Y 503.437,Z 437.558,A -85,B 0,C 180,E1 21333.672,E2 21333.672} C_VEL
LIN {X 0,Y 512.461,Z 448.664,A -85,B 0,C 180,E1 21331.286,E2 21331.286} C_VEL
LIN {X 0,Y 520.235,Z 458.793,A -85,B 0,C 180,E1 21329.367,E2 21329.367} C_VEL
LIN {X 0,Y 528.845,Z 470.027,A -85,B 0,C 180,E1 21327.399,E2 21327.399} C_VEL
LIN {X 0,Y 541.395,Z 487.245,A -85,B 0,C 180,E1 21324.755,E2 21324.755} C_VEL
LIN {X 0,Y 542.295,Z 488.859,A -85,B 0,C 180,E1 21324.566,E2 21324.566} C_VEL
LIN {X 0,Y 529.265,Z 694.502,A -85,B 0,C 180,E1 21321.235,E2 21321.235} C_VEL
LIN {X 0,Y 527.983,Z 716.444,A -85,B 0,C 180,E1 21320.882,E2 21320.882} C_VEL
LIN {X 0,Y 526.912,Z 724.128,A -85,B 0,C 180,E1 21320.846,E2 21320.846} C_VEL
LIN {X 0,Y 521.856,Z 744.674,A -85,B 0,C 180,E1 21321.055,E2 21321.055} C_VEL
LIN {X 0,Y 520.977,Z 751.266,A -85,B 0,C 180,E1 21321.012,E2 21321.012} C_VEL
LIN {X 0,Y 518.337,Z 786.331,A -85,B 0,C 180,E1 21320.379,E2 21320.379} C_VEL
LIN {X 0,Y 515.887,Z 809.19,A -85,B 0,C 180,E1 21319.82,E2 21319.82} C_VEL
LIN {X 0,Y 512.959,Z 831.4,A -85,B 0,C 180,E1 21319.145,E2 21319.145} C_VEL
LIN {X 0,Y 508.99,Z 856.629,A -85,B 0,C 180,E1 21318.211,E2 21318.211} C_VEL
LIN {X 0,Y 504.12,Z 882.063,A -85,B 0,C 180,E1 21317.049,E2 21317.049} C_VEL
LIN {X 0,Y 499.663,Z 902.808,A -85,B 0,C 180,E1 21315.934,E2 21315.934} C_VEL
LIN {X 0,Y 495.031,Z 922.49,A -85,B 0,C 180,E1 21314.717,E2 21314.717} C_VEL
LIN {X 0,Y 489.123,Z 945.51,A -85,B 0,C 180,E1 21313.081,E2 21313.081} C_VEL
LIN {X 0,Y 482.984,Z 966.986,A -85,B 0,C 180,E1 21311.284,E2 21311.284} C_VEL
LIN {X 0,Y 477.807,Z 984.23,A -85,B 0,C 180,E1 21309.639,E2 21309.639} C_VEL
LIN {X 0,Y 472.689,Z 1000.383,A -85,B 0,C 180,E1 21307.898,E2 21307.898} C_VEL
LIN {X 0,Y 467.026,Z 1017.676,A -85,B 0,C 180,E1 21305.792,E2 21305.792} C_VEL
LIN {X 0,Y 460.642,Z 1036.404,A -85,B 0,C 180,E1 21303.143,E2 21303.143} C_VEL
LIN {X 0,Y 455.771,Z 1050.479,A -85,B 0,C 180,E1 21300.855,E2 21300.855} C_VEL
LIN {X 0,Y 451.615,Z 1062.479,A -85,B 0,C 180,E1 21298.648,E2 21298.648} C_VEL
LIN {X 0,Y 447.749,Z 1073.81,A -85,B 0,C 180,E1 21296.294,E2 21296.294} C_VEL
LIN {X 0,Y 443.886,Z 1085.59,A -85,B 0,C 180,E1 21293.511,E2 21293.511} C_VEL
LIN {X 0,Y 440.09,Z 1097.65,A -85,B 0,C 180,E1 21290.156,E2 21290.156} C_VEL
LIN {X 0,Y 437.623,Z 1106.141,A -85,B 0,C 180,E1 21287.368,E2 21287.368} C_VEL
LIN {X 0,Y 435.802,Z 1113.2,A -85,B 0,C 180,E1 21284.664,E2 21284.664} C_VEL
LIN {X 0,Y 434.41,Z 1119.198,A -85,B 0,C 180,E1 21281.975,E2 21281.975} C_VEL
LIN {X 0,Y 433.522,Z 1124.077,A -85,B 0,C 180,E1 21279.366,E2 21279.366} C_VEL
LIN {X 0,Y 432.817,Z 1128.472,A -85,B 0,C 180,E1 21276.493,E2 21276.493} C_VEL
LIN {X 0,Y 432.438,Z 1132.112,A -85,B 0,C 180,E1 21273.388,E2 21273.388} C_VEL
LIN {X 0,Y 432.284,Z 1134.877,A -85,B 0,C 180,E1 21269.822,E2 21269.822} C_VEL
LIN {X 0,Y 432.201,Z 1136.097,A -85,B 0,C 180,E1 21266.668,E2 21266.668} C_VEL
LIN {X 0,Y 432.236,Z 1136.275,A -85,B 0,C 180,E1 21263.88,E2 21263.88} C_VEL
LIN {X 0,Y 432.288,Z 1135.591,A -85,B 0,C 180,E1 21261.009,E2 21261.009} C_VEL
LIN {X 0,Y 432.429,Z 1134.04,A -85,B 0,C 180,E1 21258.189,E2 21258.189} C_VEL
LIN {X 0,Y 432.711,Z 1131.534,A -85,B 0,C 180,E1 21255.274,E2 21255.274} C_VEL
LIN {X 0,Y 433.41,Z 1127.244,A -85,B 0,C 180,E1 21251.714,E2 21251.714} C_VEL
LIN {X 0,Y 434.566,Z 1121.627,A -85,B 0,C 180,E1 21248.335,E2 21248.335} C_VEL
LIN {X 0,Y 436.064,Z 1115.911,A -85,B 0,C 180,E1 21245.527,E2 21245.527} C_VEL
LIN {X 0,Y 438.045,Z 1109.21,A -85,B 0,C 180,E1 21242.748,E2 21242.748} C_VEL
LIN {X 0,Y 441.293,Z 1099.531,A -85,B 0,C 180,E1 21239.351,E2 21239.351} C_VEL
LIN {X 0,Y 445.055,Z 1088.825,A -85,B 0,C 180,E1 21236.264,E2 21236.264} C_VEL
LIN {X 0,Y 448.614,Z 1079.274,A -85,B 0,C 180,E1 21233.858,E2 21233.858} C_VEL
LIN {X 0,Y 452.879,Z 1068.007,A -85,B 0,C 180,E1 21231.365,E2 21231.365} C_VEL
LIN {X 0,Y 458.554,Z 1053.339,A -85,B 0,C 180,E1 21228.555,E2 21228.555} C_VEL
LIN {X 0,Y 464.013,Z 1038.729,A -85,B 0,C 180,E1 21226.161,E2 21226.161} C_VEL
LIN {X 0,Y 469.398,Z 1024.059,A -85,B 0,C 180,E1 21224.05,E2 21224.05} C_VEL
LIN {X 0,Y 475.915,Z 1005.793,A -85,B 0,C 180,E1 21221.757,E2 21221.757} C_VEL
LIN {X 0,Y 482.116,Z 986.89,A -85,B 0,C 180,E1 21219.736,E2 21219.736} C_VEL
LIN {X 0,Y 487.587,Z 969.292,A -85,B 0,C 180,E1 21218.085,E2 21218.085} C_VEL
LIN {X 0,Y 494.087,Z 946.634,A -85,B 0,C 180,E1 21216.252,E2 21216.252} C_VEL
LIN {X 0,Y 499.028,Z 927.662,A -85,B 0,C 180,E1 21214.927,E2 21214.927} C_VEL
LIN {X 0,Y 504.627,Z 904.615,A -85,B 0,C 180,E1 21213.524,E2 21213.524} C_VEL
LIN {X 0,Y 509.924,Z 879.528,A -85,B 0,C 180,E1 21212.244,E2 21212.244} C_VEL
LIN {X 0,Y 514.909,Z 853.814,A -85,B 0,C 180,E1 21211.139,E2 21211.139} C_VEL
LIN {X 0,Y 519.335,Z 827.722,A -85,B 0,C 180,E1 21210.224,E2 21210.224} C_VEL
LIN {X 0,Y 524.137,Z 795.697,A -85,B 0,C 180,E1 21209.343,E2 21209.343} C_VEL
LIN {X 0,Y 531.996,Z 750.75,A -85,B 0,C 180,E1 21208.359,E2 21208.359} C_VEL
LIN {X 0,Y 532.361,Z 748.88,A -85,B 0,C 180,E1 21208.307,E2 21208.307} C_VEL
LIN {X 0,Y 523.413,Z 799.791,A -85,B 0,C 180,E1 21207.202,E2 21207.202} C_VEL
LIN {X 0,Y 513.959,Z 863.637,A -85,B 0,C 180,E1 21205.778,E2 21205.778} C_VEL
LIN {X 0,Y 507.106,Z 904.87,A -85,B 0,C 180,E1 21204.661,E2 21204.661} C_VEL
LIN {X 0,Y 500.891,Z 938.835,A -85,B 0,C 180,E1 21203.559,E2 21203.559} C_VEL
LIN {X 0,Y 495.026,Z 968.948,A -85,B 0,C 180,E1 21202.352,E2 21202.352} C_VEL
LIN {X 0,Y 489.858,Z 995.312,A -85,B 0,C 180,E1 21201.108,E2 21201.108} C_VEL
LIN {X 0,Y 483.524,Z 1026.536,A -85,B 0,C 180,E1 21199.369,E2 21199.369} C_VEL
LIN {X 0,Y 478.599,Z 1049.624,A -85,B 0,C 180,E1 21197.872,E2 21197.872} C_VEL
LIN {X 0,Y 474.04,Z 1070.509,A -85,B 0,C 180,E1 21196.342,E2 21196.342} C_VEL
LIN {X 0,Y 469.431,Z 1091.071,A -85,B 0,C 180,E1 21194.649,E2 21194.649} C_VEL
LIN {X 0,Y 463.946,Z 1114.991,A -85,B 0,C 180,E1 21192.42,E2 21192.42} C_VEL
LIN {X 0,Y 458.669,Z 1137.139,A -85,B 0,C 180,E1 21190.022,E2 21190.022} C_VEL
LIN {X 0,Y 454.604,Z 1154.27,A -85,B 0,C 180,E1 21187.933,E2 21187.933} C_VEL
LIN {X 0,Y 450.952,Z 1169.689,A -85,B 0,C 180,E1 21185.828,E2 21185.828} C_VEL
LIN {X 0,Y 447.787,Z 1183.276,A -85,B 0,C 180,E1 21183.779,E2 21183.779} C_VEL
LIN {X 0,Y 444.828,Z 1196.406,A -85,B 0,C 180,E1 21181.578,E2 21181.578} C_VEL
LIN {X 0,Y 442.086,Z 1208.923,A -85,B 0,C 180,E1 21179.244,E2 21179.244} C_VEL
LIN {X 0,Y 439.717,Z 1220.147,A -85,B 0,C 180,E1 21176.905,E2 21176.905} C_VEL
LIN {X 0,Y 437.782,Z 1230.193,A -85,B 0,C 180,E1 21174.562,E2 21174.562} C_VEL
LIN {X 0,Y 436.119,Z 1239.606,A -85,B 0,C 180,E1 21172.086,E2 21172.086} C_VEL
LIN {X 0,Y 434.807,Z 1247.881,A -85,B 0,C 180,E1 21169.617,E2 21169.617} C_VEL
LIN {X 0,Y 433.792,Z 1255.6,A -85,B 0,C 180,E1 21166.946,E2 21166.946} C_VEL
LIN {X 0,Y 433.101,Z 1261.446,A -85,B 0,C 180,E1 21164.575,E2 21164.575} C_VEL
LIN {X 0,Y 432.705,Z 1266.436,A -85,B 0,C 180,E1 21162.185,E2 21162.185} C_VEL
LIN {X 0,Y 432.39,Z 1270.662,A -85,B 0,C 180,E1 21159.718,E2 21159.718} C_VEL
LIN {X 0,Y 432.284,Z 1274.099,A -85,B 0,C 180,E1 21157.115,E2 21157.115} C_VEL
LIN {X 0,Y 432.232,Z 1276.487,A -85,B 0,C 180,E1 21154.511,E2 21154.511} C_VEL
LIN {X 0,Y 432.21,Z 1277.845,A -85,B 0,C 180,E1 21151.856,E2 21151.856} C_VEL
LIN {X 0,Y 432.156,Z 1278.145,A -85,B 0,C 180,E1 21149.337,E2 21149.337} C_VEL
LIN {X 0,Y 432.186,Z 1277.42,A -85,B 0,C 180,E1 21146.684,E2 21146.684} C_VEL
LIN {X 0,Y 432.202,Z 1275.496,A -85,B 0,C 180,E1 21143.891,E2 21143.891} C_VEL
LIN {X 0,Y 432.265,Z 1272.585,A -85,B 0,C 180,E1 21141.219,E2 21141.219} C_VEL
LIN {X 0,Y 432.489,Z 1268.61,A -85,B 0,C 180,E1 21138.532,E2 21138.532} C_VEL
LIN {X 0,Y 432.891,Z 1263.543,A -85,B 0,C 180,E1 21135.828,E2 21135.828} C_VEL
LIN {X 0,Y 433.586,Z 1257.721,A -85,B 0,C 180,E1 21133.246,E2 21133.246} C_VEL
LIN {X 0,Y 434.619,Z 1250.466,A -85,B 0,C 180,E1 21130.514,E2 21130.514} C_VEL
LIN {X 0,Y 436.096,Z 1242.03,A -85,B 0,C 180,E1 21127.771,E2 21127.771} C_VEL
LIN {X 0,Y 438.092,Z 1232.169,A -85,B 0,C 180,E1 21124.973,E2 21124.973} C_VEL
LIN {X 0,Y 441.127,Z 1219.048,A -85,B 0,C 180,E1 21121.723,E2 21121.723} C_VEL
LIN {X 0,Y 444.899,Z 1204.099,A -85,B 0,C 180,E1 21118.574,E2 21118.574} C_VEL
LIN {X 0,Y 448.65,Z 1190.223,A -85,B 0,C 180,E1 21115.987,E2 21115.987} C_VEL
LIN {X 0,Y 452.797,Z 1175.596,A -85,B 0,C 180,E1 21113.558,E2 21113.558} C_VEL
LIN {X 0,Y 458.452,Z 1156.284,A -85,B 0,C 180,E1 21110.738,E2 21110.738} C_VEL
LIN {X 0,Y 464.006,Z 1137.281,A -85,B 0,C 180,E1 21108.335,E2 21108.335} C_VEL
LIN {X 0,Y 469.047,Z 1120.08,A -85,B 0,C 180,E1 21106.401,E2 21106.401} C_VEL
LIN {X 0,Y 474.261,Z 1102.009,A -85,B 0,C 180,E1 21104.593,E2 21104.593} C_VEL
LIN {X 0,Y 480.904,Z 1078.185,A -85,B 0,C 180,E1 21102.512,E2 21102.512} C_VEL
LIN {X 0,Y 486.644,Z 1056.381,A -85,B 0,C 180,E1 21100.878,E2 21100.878} C_VEL
LIN {X 0,Y 491.637,Z 1036.525,A -85,B 0,C 180,E1 21099.574,E2 21099.574} C_VEL
LIN {X 0,Y 496.37,Z 1016.341,A -85,B 0,C 180,E1 21098.409,E2 21098.409} C_VEL
LIN {X 0,Y 502.034,Z 990.563,A -85,B 0,C 180,E1 21097.138,E2 21097.138} C_VEL
LIN {X 0,Y 506.856,Z 965.3,A -85,B 0,C 180,E1 21096.126,E2 21096.126} C_VEL
LIN {X 0,Y 510.656,Z 942.889,A -85,B 0,C 180,E1 21095.384,E2 21095.384} C_VEL
LIN {X 0,Y 513.921,Z 920.754,A -85,B 0,C 180,E1 21094.787,E2 21094.787} C_VEL
LIN {X 0,Y 517.169,Z 892.592,A -85,B 0,C 180,E1 21094.178,E2 21094.178} C_VEL
LIN {X 0,Y 520.398,Z 841.815,A -85,B 0,C 180,E1 21093.327,E2 21093.327} C_VEL
LIN {X 0,Y 532.938,Z 641.734,A -85,B 0,C 180,E1 21090.051,E2 21090.051} C_VEL
LIN {X 0,Y 541.473,Z 517.061,A -85,B 0,C 180,E1 21087.972,E2 21087.972} C_VEL
LIN {X 0,Y 528.4,Z 496.374,A -85,B 0,C 180,E1 21085.05,E2 21085.05} C_VEL
LIN {X 0,Y 517.213,Z 479.497,A -85,B 0,C 180,E1 21082.296,E2 21082.296} C_VEL
LIN {X 0,Y 506.047,Z 463.224,A -85,B 0,C 180,E1 21079.267,E2 21079.267} C_VEL
LIN {X 0,Y 496.697,Z 450.295,A -85,B 0,C 180,E1 21076.46,E2 21076.46} C_VEL
LIN {X 0,Y 490.478,Z 441.627,A -85,B 0,C 180,E1 21074.401,E2 21074.401} C_VEL
LIN {X 0,Y 485.579,Z 435.046,A -85,B 0,C 180,E1 21072.668,E2 21072.668} C_VEL
LIN {X 0,Y 481.656,Z 429.715,A -85,B 0,C 180,E1 21071.192,E2 21071.192} C_VEL
LIN {X 0,Y 478.42,Z 425.438,A -85,B 0,C 180,E1 21069.929,E2 21069.929} C_VEL
LIN {X 0,Y 474.183,Z 419.661,A -85,B 0,C 180,E1 21068.122,E2 21068.122} C_VEL
LIN {X 0,Y 470.282,Z 414.611,A -85,B 0,C 180,E1 21066.409,E2 21066.409} C_VEL
LIN {X 0,Y 466.826,Z 409.716,A -85,B 0,C 180,E1 21064.699,E2 21064.699} C_VEL
LIN {X 0,Y 462.547,Z 404.334,A -85,B 0,C 180,E1 21062.54,E2 21062.54} C_VEL
LIN {X 0,Y 458.375,Z 398.809,A -85,B 0,C 180,E1 21060.125,E2 21060.125} C_VEL
LIN {X 0,Y 457.122,Z 397.203,A -85,B 0,C 180,E1 21059.373,E2 21059.373} C_VEL
LIN {X 0,Y 453.548,Z 392.381,A -85,B 0,C 180,E1 21057.041,E2 21057.041} C_VEL
LIN {X 0,Y 449.675,Z 387.631,A -85,B 0,C 180,E1 21054.257,E2 21054.257} C_VEL
LIN {X 0,Y 448.397,Z 385.586,A -85,B 0,C 180,E1 21053.213,E2 21053.213} C_VEL
LIN {X 0,Y 445.314,Z 381.8,A -85,B 0,C 180,E1 21050.566,E2 21050.566} C_VEL
LIN {X 0,Y 444.093,Z 379.64,A -85,B 0,C 180,E1 21049.361,E2 21049.361} C_VEL
LIN {X 0,Y 441.04,Z 376.002,A -85,B 0,C 180,E1 21046.162,E2 21046.162} C_VEL
LIN {X 0,Y 439.804,Z 373.844,A -85,B 0,C 180,E1 21044.568,E2 21044.568} C_VEL
LIN {X 0,Y 436.558,Z 371.645,A -85,B 0,C 180,E1 21040.464,E2 21040.464} C_VEL
LIN {X 0,Y 434.813,Z 368.88,A -85,B 0,C 180,E1 21037.131,E2 21037.131} C_VEL
LIN {X 0,Y 434.469,Z 367.59,A -85,B 0,C 180,E1 21035.373,E2 21035.373} C_VEL
LIN {X 0,Y 434.411,Z 367.134,A -85,B 0,C 180,E1 21032.144,E2 21032.144} C_VEL
LIN {X 0,Y 434.381,Z 367.118,A -85,B 0,C 180,E1 21028.498,E2 21028.498} C_VEL
LIN {X 0,Y 434.375,Z 367.109,A -85,B 0,C 180,E1 21024.705,E2 21024.705} C_VEL
LIN {X 0,Y 434.398,Z 367.103,A -85,B 0,C 180,E1 21021.068,E2 21021.068} C_VEL
LIN {X 0,Y 434.416,Z 367.102,A -85,B 0,C 180,E1 21017.414,E2 21017.414} C_VEL
LIN {X 0,Y 434.416,Z 367.304,A -85,B 0,C 180,E1 21013.669,E2 21013.669} C_VEL
LIN {X 0,Y 434.72,Z 368.539,A -85,B 0,C 180,E1 21011.424,E2 21011.424} C_VEL
LIN {X 0,Y 435.933,Z 370.886,A -85,B 0,C 180,E1 21008.937,E2 21008.937} C_VEL
LIN {X 0,Y 438.496,Z 373.145,A -85,B 0,C 180,E1 21005.505,E2 21005.505} C_VEL
LIN {X 0,Y 440.603,Z 374.451,A -85,B 0,C 180,E1 21003.311,E2 21003.311} C_VEL
LIN {X 0,Y 442.816,Z 378.336,A -85,B 0,C 180,E1 21000.901,E2 21000.901} C_VEL
LIN {X 0,Y 446.991,Z 381.395,A -85,B 0,C 180,E1 20997.583,E2 20997.583} C_VEL
LIN {X 0,Y 448.919,Z 384.943,A -85,B 0,C 180,E1 20995.948,E2 20995.948} C_VEL
LIN {X 0,Y 452.867,Z 387.904,A -85,B 0,C 180,E1 20993.451,E2 20993.451} C_VEL
LIN {X 0,Y 454.704,Z 391.222,A -85,B 0,C 180,E1 20992.213,E2 20992.213} C_VEL
LIN {X 0,Y 458.373,Z 394.014,A -85,B 0,C 180,E1 20990.234,E2 20990.234} C_VEL
LIN {X 0,Y 461.405,Z 398.511,A -85,B 0,C 180,E1 20988.575,E2 20988.575} C_VEL
LIN {X 0,Y 464.331,Z 400.956,A -85,B 0,C 180,E1 20987.191,E2 20987.191} C_VEL
LIN {X 0,Y 467.148,Z 404.921,A -85,B 0,C 180,E1 20985.837,E2 20985.837} C_VEL
LIN {X 0,Y 469.936,Z 407.379,A -85,B 0,C 180,E1 20984.667,E2 20984.667} C_VEL
LIN {X 0,Y 473.397,Z 411.858,A -85,B 0,C 180,E1 20983.186,E2 20983.186} C_VEL
LIN {X 0,Y 475.482,Z 413.893,A -85,B 0,C 180,E1 20982.386,E2 20982.386} C_VEL
LIN {X 0,Y 479.071,Z 418.326,A -85,B 0,C 180,E1 20981.009,E2 20981.009} C_VEL
LIN {X 0,Y 480.809,Z 420.243,A -85,B 0,C 180,E1 20980.373,E2 20980.373} C_VEL
LIN {X 0,Y 484.866,Z 424.957,A -85,B 0,C 180,E1 20978.959,E2 20978.959} C_VEL
LIN {X 0,Y 489.91,Z 430.966,A -85,B 0,C 180,E1 20977.291,E2 20977.291} C_VEL
LIN {X 0,Y 499.823,Z 443.143,A -85,B 0,C 180,E1 20974.302,E2 20974.302} C_VEL
LIN {X 0,Y 512.365,Z 458.811,A -85,B 0,C 180,E1 20970.95,E2 20970.95} C_VEL
LIN {X 0,Y 525.026,Z 475.641,A -85,B 0,C 180,E1 20967.926,E2 20967.926} C_VEL
LIN {X 0,Y 537.605,Z 492.99,A -85,B 0,C 180,E1 20965.212,E2 20965.212} C_VEL
LIN {X 0,Y 524.014,Z 701.096,A -85,B 0,C 180,E1 20961.824,E2 20961.824} C_VEL
LIN {X 0,Y 520.977,Z 751.266,A -85,B 0,C 180,E1 20961.012,E2 20961.012} C_VEL
LIN {X 0,Y 519.866,Z 758.951,A -85,B 0,C 180,E1 20960.976,E2 20960.976} C_VEL
LIN {X 0,Y 514.453,Z 779.431,A -85,B 0,C 180,E1 20961.164,E2 20961.164} C_VEL
LIN {X 0,Y 513.384,Z 785.958,A -85,B 0,C 180,E1 20961.087,E2 20961.087} C_VEL
LIN {X 0,Y 510.771,Z 809.821,A -85,B 0,C 180,E1 20960.504,E2 20960.504} C_VEL
LIN {X 0,Y 507.712,Z 832.421,A -85,B 0,C 180,E1 20959.814,E2 20959.814} C_VEL
LIN {X 0,Y 503.478,Z 858.634,A -85,B 0,C 180,E1 20958.835,E2 20958.835} C_VEL
LIN {X 0,Y 498.62,Z 883.39,A -85,B 0,C 180,E1 20957.695,E2 20957.695} C_VEL
LIN {X 0,Y 494.211,Z 903.501,A -85,B 0,C 180,E1 20956.612,E2 20956.612} C_VEL
LIN {X 0,Y 489.445,Z 923.229,A -85,B 0,C 180,E1 20955.387,E2 20955.387} C_VEL
LIN {X 0,Y 483.316,Z 946.469,A -85,B 0,C 180,E1 20953.726,E2 20953.726} C_VEL
LIN {X 0,Y 477.039,Z 967.829,A -85,B 0,C 180,E1 20951.928,E2 20951.928} C_VEL
LIN {X 0,Y 471.822,Z 984.728,A -85,B 0,C 180,E1 20950.309,E2 20950.309} C_VEL
LIN {X 0,Y 466.822,Z 1000.186,A -85,B 0,C 180,E1 20948.647,E2 20948.647} C_VEL
LIN {X 0,Y 461.632,Z 1015.604,A -85,B 0,C 180,E1 20946.784,E2 20946.784} C_VEL
LIN {X 0,Y 455.406,Z 1033.683,A -85,B 0,C 180,E1 20944.295,E2 20944.295} C_VEL
LIN {X 0,Y 449.498,Z 1050.058,A -85,B 0,C 180,E1 20941.654,E2 20941.654} C_VEL
LIN {X 0,Y 444.954,Z 1062.72,A -85,B 0,C 180,E1 20939.33,E2 20939.33} C_VEL
LIN {X 0,Y 440.914,Z 1074.154,A -85,B 0,C 180,E1 20936.957,E2 20936.957} C_VEL
LIN {X 0,Y 437.049,Z 1085.332,A -85,B 0,C 180,E1 20934.31,E2 20934.31} C_VEL
LIN {X 0,Y 433.025,Z 1097.642,A -85,B 0,C 180,E1 20930.923,E2 20930.923} C_VEL
LIN {X 0,Y 430.112,Z 1107.118,A -85,B 0,C 180,E1 20927.791,E2 20927.791} C_VEL
LIN {X 0,Y 428.178,Z 1114.251,A -85,B 0,C 180,E1 20925.038,E2 20925.038} C_VEL
LIN {X 0,Y 426.666,Z 1120.448,A -85,B 0,C 180,E1 20922.223,E2 20922.223} C_VEL
LIN {X 0,Y 425.652,Z 1125.672,A -85,B 0,C 180,E1 20919.365,E2 20919.365} C_VEL
LIN {X 0,Y 424.869,Z 1130.689,A -85,B 0,C 180,E1 20915.947,E2 20915.947} C_VEL
LIN {X 0,Y 424.485,Z 1134.439,A -85,B 0,C 180,E1 20912.261,E2 20912.261} C_VEL
LIN {X 0,Y 424.367,Z 1136.38,A -85,B 0,C 180,E1 20909.334,E2 20909.334} C_VEL
LIN {X 0,Y 424.306,Z 1137.377,A -85,B 0,C 180,E1 20906.599,E2 20906.599} C_VEL
LIN {X 0,Y 424.341,Z 1137.576,A -85,B 0,C 180,E1 20903.902,E2 20903.902} C_VEL
LIN {X 0,Y 424.401,Z 1136.97,A -85,B 0,C 180,E1 20901.099,E2 20901.099} C_VEL
LIN {X 0,Y 424.54,Z 1135.575,A -85,B 0,C 180,E1 20898.352,E2 20898.352} C_VEL
LIN {X 0,Y 424.818,Z 1133.353,A -85,B 0,C 180,E1 20895.564,E2 20895.564} C_VEL
LIN {X 0,Y 425.334,Z 1130.11,A -85,B 0,C 180,E1 20892.629,E2 20892.629} C_VEL
LIN {X 0,Y 426.507,Z 1124.904,A -85,B 0,C 180,E1 20889.037,E2 20889.037} C_VEL
LIN {X 0,Y 428.298,Z 1118.04,A -85,B 0,C 180,E1 20885.493,E2 20885.493} C_VEL
LIN {X 0,Y 430.391,Z 1111.322,A -85,B 0,C 180,E1 20882.607,E2 20882.607} C_VEL
LIN {X 0,Y 433.11,Z 1103.464,A -85,B 0,C 180,E1 20879.735,E2 20879.735} C_VEL
LIN {X 0,Y 437.592,Z 1091.464,A -85,B 0,C 180,E1 20876.069,E2 20876.069} C_VEL
LIN {X 0,Y 441.671,Z 1080.973,A -85,B 0,C 180,E1 20873.37,E2 20873.37} C_VEL
LIN {X 0,Y 445.888,Z 1070.345,A -85,B 0,C 180,E1 20870.969,E2 20870.969} C_VEL
LIN {X 0,Y 451.783,Z 1055.858,A -85,B 0,C 180,E1 20868.122,E2 20868.122} C_VEL
LIN {X 0,Y 457.727,Z 1040.592,A -85,B 0,C 180,E1 20865.58,E2 20865.58} C_VEL
LIN {X 0,Y 463.319,Z 1025.984,A -85,B 0,C 180,E1 20863.449,E2 20863.449} C_VEL
LIN {X 0,Y 470.081,Z 1007.81,A -85,B 0,C 180,E1 20861.137,E2 20861.137} C_VEL
LIN {X 0,Y 476.521,Z 989.05,A -85,B 0,C 180,E1 20859.101,E2 20859.101} C_VEL
LIN {X 0,Y 482.404,Z 971.016,A -85,B 0,C 180,E1 20857.388,E2 20857.388} C_VEL
LIN {X 0,Y 489.165,Z 948.528,A -85,B 0,C 180,E1 20855.548,E2 20855.548} C_VEL
LIN {X 0,Y 494.347,Z 929.87,A -85,B 0,C 180,E1 20854.223,E2 20854.223} C_VEL
LIN {X 0,Y 500.444,Z 906.38,A -85,B 0,C 180,E1 20852.771,E2 20852.771} C_VEL
LIN {X 0,Y 506.594,Z 880.038,A -85,B 0,C 180,E1 20851.404,E2 20851.404} C_VEL
LIN {X 0,Y 512.391,Z 853.054,A -85,B 0,C 180,E1 20850.238,E2 20850.238} C_VEL
LIN {X 0,Y 517.565,Z 827.314,A -85,B 0,C 180,E1 20849.326,E2 20849.326} C_VEL
LIN {X 0,Y 523.457,Z 794.441,A -85,B 0,C 180,E1 20848.428,E2 20848.428} C_VEL
LIN {X 0,Y 524.404,Z 789.571,A -85,B 0,C 180,E1 20848.307,E2 20848.307} C_VEL
LIN {X 0,Y 511.451,Z 859.995,A -85,B 0,C 180,E1 20846.7,E2 20846.7} C_VEL
LIN {X 0,Y 503.357,Z 901.831,A -85,B 0,C 180,E1 20845.524,E2 20845.524} C_VEL
LIN {X 0,Y 496.05,Z 937.571,A -85,B 0,C 180,E1 20844.323,E2 20844.323} C_VEL
LIN {X 0,Y 489.673,Z 967.974,A -85,B 0,C 180,E1 20843.074,E2 20843.074} C_VEL
LIN {X 0,Y 483.175,Z 999.046,A -85,B 0,C 180,E1 20841.56,E2 20841.56} C_VEL
LIN {X 0,Y 477.306,Z 1025.99,A -85,B 0,C 180,E1 20840,E2 20840} C_VEL
LIN {X 0,Y 472.174,Z 1048.973,A -85,B 0,C 180,E1 20838.485,E2 20838.485} C_VEL
LIN {X 0,Y 467.027,Z 1071.592,A -85,B 0,C 180,E1 20836.793,E2 20836.793} C_VEL
LIN {X 0,Y 460.758,Z 1098.217,A -85,B 0,C 180,E1 20834.502,E2 20834.502} C_VEL
LIN {X 0,Y 455.856,Z 1118.44,A -85,B 0,C 180,E1 20832.498,E2 20832.498} C_VEL
LIN {X 0,Y 451.241,Z 1137.339,A -85,B 0,C 180,E1 20830.401,E2 20830.401} C_VEL
LIN {X 0,Y 446.494,Z 1156.651,A -85,B 0,C 180,E1 20827.975,E2 20827.975} C_VEL
LIN {X 0,Y 441.668,Z 1176.591,A -85,B 0,C 180,E1 20825.101,E2 20825.101} C_VEL
LIN {X 0,Y 437.817,Z 1192.59,A -85,B 0,C 180,E1 20822.458,E2 20822.458} C_VEL
LIN {X 0,Y 434.885,Z 1205.384,A -85,B 0,C 180,E1 20820.081,E2 20820.081} C_VEL
LIN {X 0,Y 432.4,Z 1217.012,A -85,B 0,C 180,E1 20817.667,E2 20817.667} C_VEL
LIN {X 0,Y 430.227,Z 1227.72,A -85,B 0,C 180,E1 20815.17,E2 20815.17} C_VEL
LIN {X 0,Y 428.447,Z 1237.31,A -85,B 0,C 180,E1 20812.648,E2 20812.648} C_VEL
LIN {X 0,Y 427.127,Z 1245.271,A -85,B 0,C 180,E1 20810.271,E2 20810.271} C_VEL
LIN {X 0,Y 426.024,Z 1253.02,A -85,B 0,C 180,E1 20807.624,E2 20807.624} C_VEL
LIN {X 0,Y 425.258,Z 1259.59,A -85,B 0,C 180,E1 20804.989,E2 20804.989} C_VEL
LIN {X 0,Y 424.792,Z 1265.069,A -85,B 0,C 180,E1 20802.354,E2 20802.354} C_VEL
LIN {X 0,Y 424.5,Z 1269.217,A -85,B 0,C 180,E1 20799.901,E2 20799.901} C_VEL
LIN {X 0,Y 424.384,Z 1272.655,A -85,B 0,C 180,E1 20797.287,E2 20797.287} C_VEL
LIN {X 0,Y 424.34,Z 1275.128,A -85,B 0,C 180,E1 20794.595,E2 20794.595} C_VEL
LIN {X 0,Y 424.319,Z 1276.522,A -85,B 0,C 180,E1 20791.89,E2 20791.89} C_VEL
LIN {X 0,Y 424.262,Z 1276.85,A -85,B 0,C 180,E1 20789.325,E2 20789.325} C_VEL
LIN {X 0,Y 424.283,Z 1276.143,A -85,B 0,C 180,E1 20786.622,E2 20786.622} C_VEL
LIN {X 0,Y 424.285,Z 1274.36,A -85,B 0,C 180,E1 20783.912,E2 20783.912} C_VEL
LIN {X 0,Y 424.33,Z 1271.32,A -85,B 0,C 180,E1 20781.053,E2 20781.053} C_VEL
LIN {X 0,Y 424.569,Z 1267.349,A -85,B 0,C 180,E1 20778.315,E2 20778.315} C_VEL
LIN {X 0,Y 424.946,Z 1262.566,A -85,B 0,C 180,E1 20775.696,E2 20775.696} C_VEL
LIN {X 0,Y 425.706,Z 1256.448,A -85,B 0,C 180,E1 20772.927,E2 20772.927} C_VEL
LIN {X 0,Y 426.775,Z 1249.175,A -85,B 0,C 180,E1 20770.14,E2 20770.14} C_VEL
LIN {X 0,Y 428.245,Z 1241.169,A -85,B 0,C 180,E1 20767.486,E2 20767.486} C_VEL
LIN {X 0,Y 430.285,Z 1231.492,A -85,B 0,C 180,E1 20764.683,E2 20764.683} C_VEL
LIN {X 0,Y 433.321,Z 1218.806,A -85,B 0,C 180,E1 20761.468,E2 20761.468} C_VEL
LIN {X 0,Y 437.404,Z 1203.355,A -85,B 0,C 180,E1 20758.126,E2 20758.126} C_VEL
LIN {X 0,Y 441.131,Z 1190.029,A -85,B 0,C 180,E1 20755.595,E2 20755.595} C_VEL
LIN {X 0,Y 445.092,Z 1176.534,A -85,B 0,C 180,E1 20753.305,E2 20753.305} C_VEL
LIN {X 0,Y 449.745,Z 1161.089,A -85,B 0,C 180,E1 20750.957,E2 20750.957} C_VEL
LIN {X 0,Y 456.119,Z 1140.352,A -85,B 0,C 180,E1 20748.188,E2 20748.188} C_VEL
LIN {X 0,Y 461.891,Z 1121.208,A -85,B 0,C 180,E1 20745.982,E2 20745.982} C_VEL
LIN {X 0,Y 467.124,Z 1103.639,A -85,B 0,C 180,E1 20744.187,E2 20744.187} C_VEL
LIN {X 0,Y 472.574,Z 1084.894,A -85,B 0,C 180,E1 20742.484,E2 20742.484} C_VEL
LIN {X 0,Y 479.26,Z 1061.027,A -85,B 0,C 180,E1 20740.588,E2 20740.588} C_VEL
LIN {X 0,Y 485.258,Z 1037.956,A -85,B 0,C 180,E1 20739.031,E2 20739.031} C_VEL
LIN {X 0,Y 490.097,Z 1017.978,A -85,B 0,C 180,E1 20737.857,E2 20737.857} C_VEL
LIN {X 0,Y 494.942,Z 996.603,A -85,B 0,C 180,E1 20736.774,E2 20736.774} C_VEL
LIN {X 0,Y 500.439,Z 970.028,A -85,B 0,C 180,E1 20735.638,E2 20735.638} C_VEL
LIN {X 0,Y 504.996,Z 944.189,A -85,B 0,C 180,E1 20734.758,E2 20734.758} C_VEL
LIN {X 0,Y 508.316,Z 922.636,A -85,B 0,C 180,E1 20734.163,E2 20734.163} C_VEL
LIN {X 0,Y 511.152,Z 900.097,A -85,B 0,C 180,E1 20733.655,E2 20733.655} C_VEL
LIN {X 0,Y 513.565,Z 871.243,A -85,B 0,C 180,E1 20733.118,E2 20733.118} C_VEL
LIN {X 0,Y 526.561,Z 668.279,A -85,B 0,C 180,E1 20729.777,E2 20729.777} C_VEL
LIN {X 0,Y 536.887,Z 521.447,A -85,B 0,C 180,E1 20727.328,E2 20727.328} C_VEL
LIN {X 0,Y 524.762,Z 502.012,A -85,B 0,C 180,E1 20724.543,E2 20724.543} C_VEL
LIN {X 0,Y 512.397,Z 483.353,A -85,B 0,C 180,E1 20721.432,E2 20721.432} C_VEL
LIN {X 0,Y 502.411,Z 468.85,A -85,B 0,C 180,E1 20718.628,E2 20718.628} C_VEL
LIN {X 0,Y 494.878,Z 458.264,A -85,B 0,C 180,E1 20716.341,E2 20716.341} C_VEL
LIN {X 0,Y 488.485,Z 449.27,A -85,B 0,C 180,E1 20714.219,E2 20714.219} C_VEL
LIN {X 0,Y 480.601,Z 438.467,A -85,B 0,C 180,E1 20711.339,E2 20711.339} C_VEL
LIN {X 0,Y 476.203,Z 432.683,A -85,B 0,C 180,E1 20709.609,E2 20709.609} C_VEL
LIN {X 0,Y 471.955,Z 426.893,A -85,B 0,C 180,E1 20707.793,E2 20707.793} C_VEL
LIN {X 0,Y 468.245,Z 422.028,A -85,B 0,C 180,E1 20706.129,E2 20706.129} C_VEL
LIN {X 0,Y 463.981,Z 416.219,A -85,B 0,C 180,E1 20704.016,E2 20704.016} C_VEL
LIN {X 0,Y 459.562,Z 410.492,A -85,B 0,C 180,E1 20701.683,E2 20701.683} C_VEL
LIN {X 0,Y 456.402,Z 406.153,A -85,B 0,C 180,E1 20699.812,E2 20699.812} C_VEL
LIN {X 0,Y 451.796,Z 400.013,A -85,B 0,C 180,E1 20696.828,E2 20696.828} C_VEL
LIN {X 0,Y 447.924,Z 395.255,A -85,B 0,C 180,E1 20694.042,E2 20694.042} C_VEL
LIN {X 0,Y 446.753,Z 393.328,A -85,B 0,C 180,E1 20693.058,E2 20693.058} C_VEL
LIN {X 0,Y 443.643,Z 389.523,A -85,B 0,C 180,E1 20690.399,E2 20690.399} C_VEL
LIN {X 0,Y 442.438,Z 387.372,A -85,B 0,C 180,E1 20689.189,E2 20689.189} C_VEL
LIN {X 0,Y 439.441,Z 383.803,A -85,B 0,C 180,E1 20686.043,E2 20686.043} C_VEL
LIN {X 0,Y 438.148,Z 381.606,A -85,B 0,C 180,E1 20684.371,E2 20684.371} C_VEL
LIN {X 0,Y 435.013,Z 379.476,A -85,B 0,C 180,E1 20680.392,E2 20680.392} C_VEL
LIN {X 0,Y 433.306,Z 376.842,A -85,B 0,C 180,E1 20677.19,E2 20677.19} C_VEL
LIN {X 0,Y 432.584,Z 375.341,A -85,B 0,C 180,E1 20675.268,E2 20675.268} C_VEL
LIN {X 0,Y 431.092,Z 374.402,A -85,B 0,C 180,E1 20671.458,E2 20671.458} C_VEL
LIN {X 0,Y 430.12,Z 373.861,A -85,B 0,C 180,E1 20667.301,E2 20667.301} C_VEL
LIN {X 0,Y 429.922,Z 373.732,A -85,B 0,C 180,E1 20663.293,E2 20663.293} C_VEL
LIN {X 0,Y 430.51,Z 374.116,A -85,B 0,C 180,E1 20658.552,E2 20658.552} C_VEL
LIN {X 0,Y 431.804,Z 374.768,A -85,B 0,C 180,E1 20654.503,E2 20654.503} C_VEL
LIN {X 0,Y 432.818,Z 375.73,A -85,B 0,C 180,E1 20652.241,E2 20652.241} C_VEL
LIN {X 0,Y 434.475,Z 378.805,A -85,B 0,C 180,E1 20648.922,E2 20648.922} C_VEL
LIN {X 0,Y 437.079,Z 381.033,A -85,B 0,C 180,E1 20645.471,E2 20645.471} C_VEL
LIN {X 0,Y 439.188,Z 382.439,A -85,B 0,C 180,E1 20643.276,E2 20643.276} C_VEL
LIN {X 0,Y 440.965,Z 385.826,A -85,B 0,C 180,E1 20641.256,E2 20641.256} C_VEL
LIN {X 0,Y 444.301,Z 388.287,A -85,B 0,C 180,E1 20638.496,E2 20638.496} C_VEL
LIN {X 0,Y 445.429,Z 389.43,A -85,B 0,C 180,E1 20637.648,E2 20637.648} C_VEL
LIN {X 0,Y 447.458,Z 392.877,A -85,B 0,C 180,E1 20635.975,E2 20635.975} C_VEL
LIN {X 0,Y 451.089,Z 395.559,A -85,B 0,C 180,E1 20633.685,E2 20633.685} C_VEL
LIN {X 0,Y 453.028,Z 398.962,A -85,B 0,C 180,E1 20632.363,E2 20632.363} C_VEL
LIN {X 0,Y 456.882,Z 402.189,A -85,B 0,C 180,E1 20630.263,E2 20630.263} C_VEL
LIN {X 0,Y 459.708,Z 406.262,A -85,B 0,C 180,E1 20628.712,E2 20628.712} C_VEL
LIN {X 0,Y 462.494,Z 408.664,A -85,B 0,C 180,E1 20627.394,E2 20627.394} C_VEL
LIN {X 0,Y 465.459,Z 412.702,A -85,B 0,C 180,E1 20625.96,E2 20625.96} C_VEL
LIN {X 0,Y 468.022,Z 415.004,A -85,B 0,C 180,E1 20624.886,E2 20624.886} C_VEL
LIN {X 0,Y 471.649,Z 419.596,A -85,B 0,C 180,E1 20623.324,E2 20623.324} C_VEL
LIN {X 0,Y 473.503,Z 421.521,A -85,B 0,C 180,E1 20622.597,E2 20622.597} C_VEL
LIN {X 0,Y 477.415,Z 426.159,A -85,B 0,C 180,E1 20621.109,E2 20621.109} C_VEL
LIN {X 0,Y 479.731,Z 429.158,A -85,B 0,C 180,E1 20620.237,E2 20620.237} C_VEL
LIN {X 0,Y 483.814,Z 433.842,A -85,B 0,C 180,E1 20618.827,E2 20618.827} C_VEL
LIN {X 0,Y 489.051,Z 440.215,A -85,B 0,C 180,E1 20617.105,E2 20617.105} C_VEL
LIN {X 0,Y 494.531,Z 446.912,A -85,B 0,C 180,E1 20615.424,E2 20615.424} C_VEL
LIN {X 0,Y 501.8,Z 455.965,A -85,B 0,C 180,E1 20613.34,E2 20613.34} C_VEL
LIN {X 0,Y 511.013,Z 467.665,A -85,B 0,C 180,E1 20610.924,E2 20610.924} C_VEL
LIN {X 0,Y 522.195,Z 482.607,A -85,B 0,C 180,E1 20608.228,E2 20608.228} C_VEL
LIN {X 0,Y 532.957,Z 497.653,A -85,B 0,C 180,E1 20605.86,E2 20605.86} C_VEL
LIN {X 0,Y 519.428,Z 697.851,A -85,B 0,C 180,E1 20602.584,E2 20602.584} C_VEL
LIN {X 0,Y 514.088,Z 778.502,A -85,B 0,C 180,E1 20601.239,E2 20601.239} C_VEL
LIN {X 0,Y 513.384,Z 785.958,A -85,B 0,C 180,E1 20601.087,E2 20601.087} C_VEL
LIN {X 0,Y 511.936,Z 793.561,A -85,B 0,C 180,E1 20601.014,E2 20601.014} C_VEL
LIN {X 0,Y 506.276,Z 811.709,A -85,B 0,C 180,E1 20601.068,E2 20601.068} C_VEL
LIN {X 0,Y 504.641,Z 819.225,A -85,B 0,C 180,E1 20600.951,E2 20600.951} C_VEL
LIN {X 0,Y 504.502,Z 820.294,A -85,B 0,C 180,E1 20600.922,E2 20600.922} C_VEL
LIN {X 0,Y 500.399,Z 846.693,A -85,B 0,C 180,E1 20600.021,E2 20600.021} C_VEL
LIN {X 0,Y 496.431,Z 868.524,A -85,B 0,C 180,E1 20599.119,E2 20599.119} C_VEL
LIN {X 0,Y 492.095,Z 889.592,A -85,B 0,C 180,E1 20598.098,E2 20598.098} C_VEL
LIN {X 0,Y 486.12,Z 915.289,A -85,B 0,C 180,E1 20596.633,E2 20596.633} C_VEL
LIN {X 0,Y 480.409,Z 936.97,A -85,B 0,C 180,E1 20595.167,E2 20595.167} C_VEL
LIN {X 0,Y 475.03,Z 955.799,A -85,B 0,C 180,E1 20593.707,E2 20593.707} C_VEL
LIN {X 0,Y 469.147,Z 975.103,A -85,B 0,C 180,E1 20591.999,E2 20591.999} C_VEL
LIN {X 0,Y 461.74,Z 997.767,A -85,B 0,C 180,E1 20589.662,E2 20589.662} C_VEL
LIN {X 0,Y 456.067,Z 1014.219,A -85,B 0,C 180,E1 20587.699,E2 20587.699} C_VEL
LIN {X 0,Y 450.844,Z 1028.936,A -85,B 0,C 180,E1 20585.717,E2 20585.717} C_VEL
LIN {X 0,Y 445.634,Z 1043.242,A -85,B 0,C 180,E1 20583.542,E2 20583.542} C_VEL
LIN {X 0,Y 439.512,Z 1059.983,A -85,B 0,C 180,E1 20580.614,E2 20580.614} C_VEL
LIN {X 0,Y 434.418,Z 1073.643,A -85,B 0,C 180,E1 20577.811,E2 20577.811} C_VEL
LIN {X 0,Y 430.531,Z 1084.374,A -85,B 0,C 180,E1 20575.301,E2 20575.301} C_VEL
LIN {X 0,Y 427.187,Z 1094.012,A -85,B 0,C 180,E1 20572.733,E2 20572.733} C_VEL
LIN {X 0,Y 424.185,Z 1103.114,A -85,B 0,C 180,E1 20569.946,E2 20569.946} C_VEL
LIN {X 0,Y 421.231,Z 1113.032,A -85,B 0,C 180,E1 20566.385,E2 20566.385} C_VEL
LIN {X 0,Y 419.146,Z 1120.805,A -85,B 0,C 180,E1 20562.916,E2 20562.916} C_VEL
LIN {X 0,Y 417.998,Z 1126.125,A -85,B 0,C 180,E1 20560.052,E2 20560.052} C_VEL
LIN {X 0,Y 417.174,Z 1130.657,A -85,B 0,C 180,E1 20557.048,E2 20557.048} C_VEL
LIN {X 0,Y 416.762,Z 1134.061,A -85,B 0,C 180,E1 20554.136,E2 20554.136} C_VEL
LIN {X 0,Y 416.522,Z 1137.164,A -85,B 0,C 180,E1 20550.433,E2 20550.433} C_VEL
LIN {X 0,Y 416.396,Z 1138.588,A -85,B 0,C 180,E1 20546.991,E2 20546.991} C_VEL
LIN {X 0,Y 416.44,Z 1138.897,A -85,B 0,C 180,E1 20544.091,E2 20544.091} C_VEL
LIN {X 0,Y 416.517,Z 1138.333,A -85,B 0,C 180,E1 20541.106,E2 20541.106} C_VEL
LIN {X 0,Y 416.671,Z 1136.999,A -85,B 0,C 180,E1 20538.322,E2 20538.322} C_VEL
LIN {X 0,Y 416.978,Z 1134.771,A -85,B 0,C 180,E1 20535.43,E2 20535.43} C_VEL
LIN {X 0,Y 417.547,Z 1131.565,A -85,B 0,C 180,E1 20532.446,E2 20532.446} C_VEL
LIN {X 0,Y 418.789,Z 1126.409,A -85,B 0,C 180,E1 20528.79,E2 20528.79} C_VEL
LIN {X 0,Y 420.709,Z 1119.602,A -85,B 0,C 180,E1 20525.182,E2 20525.182} C_VEL
LIN {X 0,Y 422.874,Z 1113.062,A -85,B 0,C 180,E1 20522.304,E2 20522.304} C_VEL
LIN {X 0,Y 425.941,Z 1104.727,A -85,B 0,C 180,E1 20519.193,E2 20519.193} C_VEL
LIN {X 0,Y 430.497,Z 1093.152,A -85,B 0,C 180,E1 20515.604,E2 20515.604} C_VEL
LIN {X 0,Y 434.557,Z 1083.252,A -85,B 0,C 180,E1 20512.995,E2 20512.995} C_VEL
LIN {X 0,Y 439.43,Z 1071.556,A -85,B 0,C 180,E1 20510.306,E2 20510.306} C_VEL
LIN {X 0,Y 445.744,Z 1056.628,A -85,B 0,C 180,E1 20507.362,E2 20507.362} C_VEL
LIN {X 0,Y 451.821,Z 1041.738,A -85,B 0,C 180,E1 20504.862,E2 20504.862} C_VEL
LIN {X 0,Y 457.343,Z 1027.915,A -85,B 0,C 180,E1 20502.823,E2 20502.823} C_VEL
LIN {X 0,Y 463.977,Z 1010.909,A -85,B 0,C 180,E1 20500.617,E2 20500.617} C_VEL
LIN {X 0,Y 471.033,Z 991.356,A -85,B 0,C 180,E1 20498.455,E2 20498.455} C_VEL
LIN {X 0,Y 477.152,Z 973.547,A -85,B 0,C 180,E1 20496.733,E2 20496.733} C_VEL
LIN {X 0,Y 484.202,Z 951.438,A -85,B 0,C 180,E1 20494.89,E2 20494.89} C_VEL
LIN {X 0,Y 490.09,Z 931.703,A -85,B 0,C 180,E1 20493.461,E2 20493.461} C_VEL
LIN {X 0,Y 497.243,Z 906.056,A -85,B 0,C 180,E1 20491.865,E2 20491.865} C_VEL
LIN {X 0,Y 504.223,Z 879.641,A -85,B 0,C 180,E1 20490.476,E2 20490.476} C_VEL
LIN {X 0,Y 511.425,Z 850.645,A -85,B 0,C 180,E1 20489.228,E2 20489.228} C_VEL
LIN {X 0,Y 516.907,Z 826.695,A -85,B 0,C 180,E1 20488.39,E2 20488.39} C_VEL
LIN {X 0,Y 506.615,Z 871.737,A -85,B 0,C 180,E1 20487.259,E2 20487.259} C_VEL
LIN {X 0,Y 496.239,Z 916.503,A -85,B 0,C 180,E1 20485.855,E2 20485.855} C_VEL
LIN {X 0,Y 488.736,Z 949.149,A -85,B 0,C 180,E1 20484.621,E2 20484.621} C_VEL
LIN {X 0,Y 481.364,Z 981.181,A -85,B 0,C 180,E1 20483.157,E2 20483.157} C_VEL
LIN {X 0,Y 474.96,Z 1009.3,A -85,B 0,C 180,E1 20481.645,E2 20481.645} C_VEL
LIN {X 0,Y 467.904,Z 1039.865,A -85,B 0,C 180,E1 20479.719,E2 20479.719} C_VEL
LIN {X 0,Y 462.218,Z 1063.655,A -85,B 0,C 180,E1 20477.978,E2 20477.978} C_VEL
LIN {X 0,Y 457.21,Z 1084.173,A -85,B 0,C 180,E1 20476.285,E2 20476.285} C_VEL
LIN {X 0,Y 452.031,Z 1105.056,A -85,B 0,C 180,E1 20474.345,E2 20474.345} C_VEL
LIN {X 0,Y 445.715,Z 1130.138,A -85,B 0,C 180,E1 20471.666,E2 20471.666} C_VEL
LIN {X 0,Y 440.764,Z 1149.666,A -85,B 0,C 180,E1 20469.265,E2 20469.265} C_VEL
LIN {X 0,Y 436.288,Z 1167.242,A -85,B 0,C 180,E1 20466.821,E2 20466.821} C_VEL
LIN {X 0,Y 431.554,Z 1186.414,A -85,B 0,C 180,E1 20463.784,E2 20463.784} C_VEL
LIN {X 0,Y 427.63,Z 1202.574,A -85,B 0,C 180,E1 20460.801,E2 20460.801} C_VEL
LIN {X 0,Y 424.873,Z 1214.87,A -85,B 0,C 180,E1 20458.231,E2 20458.231} C_VEL
LIN {X 0,Y 422.579,Z 1225.882,A -85,B 0,C 180,E1 20455.643,E2 20455.643} C_VEL
LIN {X 0,Y 420.715,Z 1235.482,A -85,B 0,C 180,E1 20453.088,E2 20453.088} C_VEL
LIN {X 0,Y 419.267,Z 1243.993,A -85,B 0,C 180,E1 20450.522,E2 20450.522} C_VEL
LIN {X 0,Y 418.139,Z 1251.598,A -85,B 0,C 180,E1 20447.873,E2 20447.873} C_VEL
LIN {X 0,Y 417.393,Z 1258.015,A -85,B 0,C 180,E1 20445.278,E2 20445.278} C_VEL
LIN {X 0,Y 416.871,Z 1263.81,A -85,B 0,C 180,E1 20442.466,E2 20442.466} C_VEL
LIN {X 0,Y 416.572,Z 1268.192,A -85,B 0,C 180,E1 20439.812,E2 20439.812} C_VEL
LIN {X 0,Y 416.478,Z 1271.541,A -85,B 0,C 180,E1 20437.172,E2 20437.172} C_VEL
LIN {X 0,Y 416.443,Z 1273.872,A -85,B 0,C 180,E1 20434.544,E2 20434.544} C_VEL
LIN {X 0,Y 416.427,Z 1275.206,A -85,B 0,C 180,E1 20431.926,E2 20431.926} C_VEL
LIN {X 0,Y 416.368,Z 1275.554,A -85,B 0,C 180,E1 20429.312,E2 20429.312} C_VEL
LIN {X 0,Y 416.379,Z 1274.866,A -85,B 0,C 180,E1 20426.558,E2 20426.558} C_VEL
LIN {X 0,Y 416.371,Z 1273.095,A -85,B 0,C 180,E1 20423.796,E2 20423.796} C_VEL
LIN {X 0,Y 416.395,Z 1270.246,A -85,B 0,C 180,E1 20421.02,E2 20421.02} C_VEL
LIN {X 0,Y 416.65,Z 1266.097,A -85,B 0,C 180,E1 20418.09,E2 20418.09} C_VEL
LIN {X 0,Y 417.068,Z 1261.019,A -85,B 0,C 180,E1 20415.278,E2 20415.278} C_VEL
LIN {X 0,Y 417.858,Z 1254.83,A -85,B 0,C 180,E1 20412.452,E2 20412.452} C_VEL
LIN {X 0,Y 418.973,Z 1247.728,A -85,B 0,C 180,E1 20409.703,E2 20409.703} C_VEL
LIN {X 0,Y 420.493,Z 1239.825,A -85,B 0,C 180,E1 20407.047,E2 20407.047} C_VEL
LIN {X 0,Y 422.65,Z 1230.141,A -85,B 0,C 180,E1 20404.196,E2 20404.196} C_VEL
LIN {X 0,Y 425.995,Z 1216.842,A -85,B 0,C 180,E1 20400.777,E2 20400.777} C_VEL
LIN {X 0,Y 430.11,Z 1201.857,A -85,B 0,C 180,E1 20397.52,E2 20397.52} C_VEL
LIN {X 0,Y 433.954,Z 1188.689,A -85,B 0,C 180,E1 20394.99,E2 20394.99} C_VEL
LIN {X 0,Y 438.174,Z 1174.935,A -85,B 0,C 180,E1 20392.628,E2 20392.628} C_VEL
LIN {X 0,Y 443.557,Z 1157.908,A -85,B 0,C 180,E1 20390.025,E2 20390.025} C_VEL
LIN {X 0,Y 450.128,Z 1136.985,A -85,B 0,C 180,E1 20387.265,E2 20387.265} C_VEL
LIN {X 0,Y 455.672,Z 1119.27,A -85,B 0,C 180,E1 20385.222,E2 20385.222} C_VEL
LIN {X 0,Y 461.12,Z 1101.637,A -85,B 0,C 180,E1 20383.414,E2 20383.414} C_VEL
LIN {X 0,Y 467.274,Z 1081.155,A -85,B 0,C 180,E1 20381.556,E2 20381.556} C_VEL
LIN {X 0,Y 474.288,Z 1056.336,A -85,B 0,C 180,E1 20379.628,E2 20379.628} C_VEL
LIN {X 0,Y 479.881,Z 1035.36,A -85,B 0,C 180,E1 20378.231,E2 20378.231} C_VEL
LIN {X 0,Y 484.884,Z 1015.21,A -85,B 0,C 180,E1 20377.058,E2 20377.058} C_VEL
LIN {X 0,Y 490.43,Z 991.324,A -85,B 0,C 180,E1 20375.864,E2 20375.864} C_VEL
LIN {X 0,Y 495.948,Z 964.335,A -85,B 0,C 180,E1 20374.759,E2 20374.759} C_VEL
LIN {X 0,Y 500.011,Z 941.822,A -85,B 0,C 180,E1 20374.008,E2 20374.008} C_VEL
LIN {X 0,Y 503.425,Z 920.029,A -85,B 0,C 180,E1 20373.413,E2 20373.413} C_VEL
LIN {X 0,Y 506.767,Z 893.218,A -85,B 0,C 180,E1 20372.818,E2 20372.818} C_VEL
LIN {X 0,Y 509.679,Z 852.353,A -85,B 0,C 180,E1 20372.11,E2 20372.11} C_VEL
LIN {X 0,Y 524.16,Z 637.306,A -85,B 0,C 180,E1 20368.542,E2 20368.542} C_VEL
LIN {X 0,Y 532.335,Z 525.825,A -85,B 0,C 180,E1 20366.674,E2 20366.674} C_VEL
LIN {X 0,Y 521.389,Z 508.197,A -85,B 0,C 180,E1 20364.109,E2 20364.109} C_VEL
LIN {X 0,Y 509.735,Z 490.394,A -85,B 0,C 180,E1 20361.127,E2 20361.127} C_VEL
LIN {X 0,Y 499.8,Z 475.869,A -85,B 0,C 180,E1 20358.306,E2 20358.306} C_VEL
LIN {X 0,Y 492.317,Z 465.175,A -85,B 0,C 180,E1 20355.974,E2 20355.974} C_VEL
LIN {X 0,Y 485.524,Z 455.68,A -85,B 0,C 180,E1 20353.7,E2 20353.7} C_VEL
LIN {X 0,Y 478.474,Z 445.88,A -85,B 0,C 180,E1 20351.085,E2 20351.085} C_VEL
LIN {X 0,Y 474.001,Z 439.926,A -85,B 0,C 180,E1 20349.287,E2 20349.287} C_VEL
LIN {X 0,Y 469.741,Z 434.121,A -85,B 0,C 180,E1 20347.461,E2 20347.461} C_VEL
LIN {X 0,Y 466.219,Z 429.443,A -85,B 0,C 180,E1 20345.847,E2 20345.847} C_VEL
LIN {X 0,Y 461.913,Z 423.614,A -85,B 0,C 180,E1 20343.715,E2 20343.715} C_VEL
LIN {X 0,Y 457.71,Z 418.048,A -85,B 0,C 180,E1 20341.44,E2 20341.44} C_VEL
LIN {X 0,Y 454.443,Z 413.497,A -85,B 0,C 180,E1 20339.496,E2 20339.496} C_VEL
LIN {X 0,Y 450.127,Z 407.824,A -85,B 0,C 180,E1 20336.689,E2 20336.689} C_VEL
LIN {X 0,Y 446.103,Z 402.735,A -85,B 0,C 180,E1 20333.759,E2 20333.759} C_VEL
LIN {X 0,Y 444.924,Z 400.91,A -85,B 0,C 180,E1 20332.77,E2 20332.77} C_VEL
LIN {X 0,Y 441.893,Z 397.116,A -85,B 0,C 180,E1 20330.163,E2 20330.163} C_VEL
LIN {X 0,Y 440.787,Z 395.107,A -85,B 0,C 180,E1 20329.015,E2 20329.015} C_VEL
LIN {X 0,Y 437.789,Z 391.496,A -85,B 0,C 180,E1 20325.855,E2 20325.855} C_VEL
LIN {X 0,Y 436.611,Z 389.448,A -85,B 0,C 180,E1 20324.322,E2 20324.322} C_VEL
LIN {X 0,Y 433.428,Z 387.258,A -85,B 0,C 180,E1 20320.257,E2 20320.257} C_VEL
LIN {X 0,Y 431.76,Z 384.668,A -85,B 0,C 180,E1 20317.104,E2 20317.104} C_VEL
LIN {X 0,Y 431.038,Z 383.17,A -85,B 0,C 180,E1 20315.173,E2 20315.173} C_VEL
LIN {X 0,Y 429.486,Z 382.215,A -85,B 0,C 180,E1 20311.189,E2 20311.189} C_VEL
LIN {X 0,Y 428.586,Z 381.709,A -85,B 0,C 180,E1 20307.072,E2 20307.072} C_VEL
LIN {X 0,Y 428.471,Z 381.654,A -85,B 0,C 180,E1 20302.813,E2 20302.813} C_VEL
LIN {X 0,Y 429.089,Z 382.011,A -85,B 0,C 180,E1 20298.206,E2 20298.206} C_VEL
LIN {X 0,Y 430.489,Z 382.715,A -85,B 0,C 180,E1 20294.134,E2 20294.134} C_VEL
LIN {X 0,Y 431.412,Z 383.793,A -85,B 0,C 180,E1 20292.052,E2 20292.052} C_VEL
LIN {X 0,Y 433.019,Z 386.723,A -85,B 0,C 180,E1 20288.906,E2 20288.906} C_VEL
LIN {X 0,Y 435.76,Z 388.967,A -85,B 0,C 180,E1 20285.326,E2 20285.326} C_VEL
LIN {X 0,Y 437.63,Z 390.258,A -85,B 0,C 180,E1 20283.41,E2 20283.41} C_VEL
LIN {X 0,Y 439.439,Z 393.676,A -85,B 0,C 180,E1 20281.327,E2 20281.327} C_VEL
LIN {X 0,Y 442.802,Z 396.134,A -85,B 0,C 180,E1 20278.55,E2 20278.55} C_VEL
LIN {X 0,Y 443.719,Z 397.123,A -85,B 0,C 180,E1 20277.845,E2 20277.845} C_VEL
LIN {X 0,Y 445.733,Z 400.517,A -85,B 0,C 180,E1 20276.194,E2 20276.194} C_VEL
LIN {X 0,Y 449.385,Z 403.364,A -85,B 0,C 180,E1 20273.867,E2 20273.867} C_VEL
LIN {X 0,Y 451.568,Z 406.938,A -85,B 0,C 180,E1 20272.386,E2 20272.386} C_VEL
LIN {X 0,Y 455.136,Z 409.953,A -85,B 0,C 180,E1 20270.445,E2 20270.445} C_VEL
LIN {X 0,Y 458.013,Z 414.01,A -85,B 0,C 180,E1 20268.85,E2 20268.85} C_VEL
LIN {X 0,Y 460.673,Z 416.363,A -85,B 0,C 180,E1 20267.596,E2 20267.596} C_VEL
LIN {X 0,Y 463.932,Z 420.626,A -85,B 0,C 180,E1 20266.014,E2 20266.014} C_VEL
LIN {X 0,Y 466.061,Z 422.604,A -85,B 0,C 180,E1 20265.107,E2 20265.107} C_VEL
LIN {X 0,Y 469.882,Z 427.313,A -85,B 0,C 180,E1 20263.472,E2 20263.472} C_VEL
LIN {X 0,Y 471.55,Z 429.166,A -85,B 0,C 180,E1 20262.802,E2 20262.802} C_VEL
LIN {X 0,Y 475.576,Z 433.825,A -85,B 0,C 180,E1 20261.276,E2 20261.276} C_VEL
LIN {X 0,Y 481.88,Z 441.597,A -85,B 0,C 180,E1 20258.997,E2 20258.997} C_VEL
LIN {X 0,Y 486.831,Z 447.58,A -85,B 0,C 180,E1 20257.369,E2 20257.369} C_VEL
LIN {X 0,Y 494.61,Z 457.055,A -85,B 0,C 180,E1 20254.987,E2 20254.987} C_VEL
LIN {X 0,Y 507.13,Z 473.035,A -85,B 0,C 180,E1 20251.54,E2 20251.54} C_VEL
LIN {X 0,Y 519.241,Z 489.379,A -85,B 0,C 180,E1 20248.566,E2 20248.566} C_VEL
LIN {X 0,Y 528.371,Z 502.225,A -85,B 0,C 180,E1 20246.52,E2 20246.52} C_VEL
LIN {X 0,Y 513.977,Z 708.198,A -85,B 0,C 180,E1 20243.129,E2 20243.129} C_VEL
LIN {X 0,Y 509.112,Z 779.223,A -85,B 0,C 180,E1 20241.936,E2 20241.936} C_VEL
LIN {X 0,Y 506.059,Z 807.883,A -85,B 0,C 180,E1 20241.271,E2 20241.271} C_VEL
LIN {X 0,Y 504.502,Z 820.294,A -85,B 0,C 180,E1 20240.922,E2 20240.922} C_VEL
LIN {X 0,Y 502.9,Z 827.789,A -85,B 0,C 180,E1 20240.78,E2 20240.78} C_VEL
LIN {X 0,Y 496.041,Z 846.7,A -85,B 0,C 180,E1 20240.66,E2 20240.66} C_VEL
LIN {X 0,Y 494.121,Z 854.004,A -85,B 0,C 180,E1 20240.469,E2 20240.469} C_VEL
LIN {X 0,Y 488.834,Z 881.02,A -85,B 0,C 180,E1 20239.273,E2 20239.273} C_VEL
LIN {X 0,Y 483.697,Z 903.539,A -85,B 0,C 180,E1 20238.07,E2 20238.07} C_VEL
LIN {X 0,Y 478.964,Z 922.405,A -85,B 0,C 180,E1 20236.909,E2 20236.909} C_VEL
LIN {X 0,Y 473.75,Z 941.429,A -85,B 0,C 180,E1 20235.579,E2 20235.579} C_VEL
LIN {X 0,Y 467.171,Z 963.83,A -85,B 0,C 180,E1 20233.781,E2 20233.781} C_VEL
LIN {X 0,Y 460.524,Z 984.319,A -85,B 0,C 180,E1 20231.847,E2 20231.847} C_VEL
LIN {X 0,Y 454.916,Z 1000.704,A -85,B 0,C 180,E1 20230.082,E2 20230.082} C_VEL
LIN {X 0,Y 449.359,Z 1016.307,A -85,B 0,C 180,E1 20228.186,E2 20228.186} C_VEL
LIN {X 0,Y 443.892,Z 1031.222,A -85,B 0,C 180,E1 20226.141,E2 20226.141} C_VEL
LIN {X 0,Y 437.474,Z 1048.486,A -85,B 0,C 180,E1 20223.446,E2 20223.446} C_VEL
LIN {X 0,Y 431.482,Z 1064.038,A -85,B 0,C 180,E1 20220.576,E2 20220.576} C_VEL
LIN {X 0,Y 427.135,Z 1075.386,A -85,B 0,C 180,E1 20218.186,E2 20218.186} C_VEL
LIN {X 0,Y 423.31,Z 1085.56,A -85,B 0,C 180,E1 20215.764,E2 20215.764} C_VEL
LIN {X 0,Y 420.007,Z 1094.695,A -85,B 0,C 180,E1 20213.307,E2 20213.307} C_VEL
LIN {X 0,Y 416.982,Z 1103.485,A -85,B 0,C 180,E1 20210.613,E2 20210.613} C_VEL
LIN {X 0,Y 414.314,Z 1111.768,A -85,B 0,C 180,E1 20207.676,E2 20207.676} C_VEL
LIN {X 0,Y 411.76,Z 1120.748,A -85,B 0,C 180,E1 20203.846,E2 20203.846} C_VEL
LIN {X 0,Y 410.283,Z 1126.978,A -85,B 0,C 180,E1 20200.505,E2 20200.505} C_VEL
LIN {X 0,Y 409.422,Z 1131.349,A -85,B 0,C 180,E1 20197.63,E2 20197.63} C_VEL
LIN {X 0,Y 408.943,Z 1134.825,A -85,B 0,C 180,E1 20194.729,E2 20194.729} C_VEL
LIN {X 0,Y 408.674,Z 1137.488,A -85,B 0,C 180,E1 20191.738,E2 20191.738} C_VEL
LIN {X 0,Y 408.562,Z 1139.21,A -85,B 0,C 180,E1 20188.821,E2 20188.821} C_VEL
LIN {X 0,Y 408.546,Z 1140.133,A -85,B 0,C 180,E1 20185.671,E2 20185.671} C_VEL
LIN {X 0,Y 408.629,Z 1139.951,A -85,B 0,C 180,E1 20181.835,E2 20181.835} C_VEL
LIN {X 0,Y 408.778,Z 1138.569,A -85,B 0,C 180,E1 20178.541,E2 20178.541} C_VEL
LIN {X 0,Y 409.098,Z 1136.459,A -85,B 0,C 180,E1 20175.596,E2 20175.596} C_VEL
LIN {X 0,Y 409.624,Z 1133.546,A -85,B 0,C 180,E1 20172.691,E2 20172.691} C_VEL
LIN {X 0,Y 410.612,Z 1129.574,A -85,B 0,C 180,E1 20169.673,E2 20169.673} C_VEL
LIN {X 0,Y 412.275,Z 1123.954,A -85,B 0,C 180,E1 20166.266,E2 20166.266} C_VEL
LIN {X 0,Y 414.956,Z 1116.018,A -85,B 0,C 180,E1 20162.486,E2 20162.486} C_VEL
LIN {X 0,Y 417.897,Z 1108.283,A -85,B 0,C 180,E1 20159.452,E2 20159.452} C_VEL
LIN {X 0,Y 421.728,Z 1098.95,A -85,B 0,C 180,E1 20156.33,E2 20156.33} C_VEL
LIN {X 0,Y 427.248,Z 1086.084,A -85,B 0,C 180,E1 20152.74,E2 20152.74} C_VEL
LIN {X 0,Y 432.011,Z 1075.133,A -85,B 0,C 180,E1 20150.138,E2 20150.138} C_VEL
LIN {X 0,Y 437.444,Z 1062.849,A -85,B 0,C 180,E1 20147.593,E2 20147.593} C_VEL
LIN {X 0,Y 444.728,Z 1046.061,A -85,B 0,C 180,E1 20144.615,E2 20144.615} C_VEL
LIN {X 0,Y 450.712,Z 1031.787,A -85,B 0,C 180,E1 20142.44,E2 20142.44} C_VEL
LIN {X 0,Y 457.552,Z 1015.008,A -85,B 0,C 180,E1 20140.201,E2 20140.201} C_VEL
LIN {X 0,Y 465.063,Z 995.436,A -85,B 0,C 180,E1 20137.965,E2 20137.965} C_VEL
LIN {X 0,Y 471.39,Z 978.056,A -85,B 0,C 180,E1 20136.233,E2 20136.233} C_VEL
LIN {X 0,Y 479.182,Z 955.355,A -85,B 0,C 180,E1 20134.277,E2 20134.277} C_VEL
LIN {X 0,Y 486.315,Z 933.253,A -85,B 0,C 180,E1 20132.643,E2 20132.643} C_VEL
LIN {X 0,Y 493.954,Z 908.39,A -85,B 0,C 180,E1 20131.066,E2 20131.066} C_VEL
LIN {X 0,Y 502.384,Z 880.355,A -85,B 0,C 180,E1 20129.567,E2 20129.567} C_VEL
LIN {X 0,Y 509.092,Z 857.704,A -85,B 0,C 180,E1 20128.553,E2 20128.553} C_VEL
LIN {X 0,Y 498.222,Z 896.628,A -85,B 0,C 180,E1 20127.393,E2 20127.393} C_VEL
LIN {X 0,Y 487.501,Z 936.311,A -85,B 0,C 180,E1 20125.948,E2 20125.948} C_VEL
LIN {X 0,Y 478.329,Z 972.369,A -85,B 0,C 180,E1 20124.341,E2 20124.341} C_VEL
LIN {X 0,Y 470.987,Z 1001.977,A -85,B 0,C 180,E1 20122.759,E2 20122.759} C_VEL
LIN {X 0,Y 463.738,Z 1031.807,A -85,B 0,C 180,E1 20120.914,E2 20120.914} C_VEL
LIN {X 0,Y 456.874,Z 1059.083,A -85,B 0,C 180,E1 20118.933,E2 20118.933} C_VEL
LIN {X 0,Y 451.587,Z 1079.854,A -85,B 0,C 180,E1 20117.222,E2 20117.222} C_VEL
LIN {X 0,Y 446.505,Z 1099.504,A -85,B 0,C 180,E1 20115.407,E2 20115.407} C_VEL
LIN {X 0,Y 441.327,Z 1119.319,A -85,B 0,C 180,E1 20113.352,E2 20113.352} C_VEL
LIN {X 0,Y 435.234,Z 1142.317,A -85,B 0,C 180,E1 20110.634,E2 20110.634} C_VEL
LIN {X 0,Y 430.165,Z 1161.576,A -85,B 0,C 180,E1 20108.002,E2 20108.002} C_VEL
LIN {X 0,Y 425.873,Z 1178.106,A -85,B 0,C 180,E1 20105.441,E2 20105.441} C_VEL
LIN {X 0,Y 422.095,Z 1192.917,A -85,B 0,C 180,E1 20102.851,E2 20102.851} C_VEL
LIN {X 0,Y 418.285,Z 1209.02,A -85,B 0,C 180,E1 20099.658,E2 20099.658} C_VEL
LIN {X 0,Y 415.096,Z 1223.176,A -85,B 0,C 180,E1 20096.352,E2 20096.352} C_VEL
LIN {X 0,Y 413.001,Z 1233.686,A -85,B 0,C 180,E1 20093.545,E2 20093.545} C_VEL
LIN {X 0,Y 411.492,Z 1242.25,A -85,B 0,C 180,E1 20090.928,E2 20090.928} C_VEL
LIN {X 0,Y 410.332,Z 1249.72,A -85,B 0,C 180,E1 20088.321,E2 20088.321} C_VEL
LIN {X 0,Y 409.53,Z 1256.44,A -85,B 0,C 180,E1 20085.579,E2 20085.579} C_VEL
LIN {X 0,Y 408.987,Z 1262.029,A -85,B 0,C 180,E1 20082.854,E2 20082.854} C_VEL
LIN {X 0,Y 408.694,Z 1266.549,A -85,B 0,C 180,E1 20080.145,E2 20080.145} C_VEL
LIN {X 0,Y 408.569,Z 1270.163,A -85,B 0,C 180,E1 20077.311,E2 20077.311} C_VEL
LIN {X 0,Y 408.545,Z 1272.541,A -85,B 0,C 180,E1 20074.632,E2 20074.632} C_VEL
LIN {X 0,Y 408.529,Z 1273.946,A -85,B 0,C 180,E1 20071.823,E2 20071.823} C_VEL
LIN {X 0,Y 408.471,Z 1274.263,A -85,B 0,C 180,E1 20069.158,E2 20069.158} C_VEL
LIN {X 0,Y 408.473,Z 1273.538,A -85,B 0,C 180,E1 20066.351,E2 20066.351} C_VEL
LIN {X 0,Y 408.452,Z 1271.722,A -85,B 0,C 180,E1 20063.534,E2 20063.534} C_VEL
LIN {X 0,Y 408.466,Z 1268.819,A -85,B 0,C 180,E1 20060.702,E2 20060.702} C_VEL
LIN {X 0,Y 408.726,Z 1264.843,A -85,B 0,C 180,E1 20057.855,E2 20057.855} C_VEL
LIN {X 0,Y 409.168,Z 1259.744,A -85,B 0,C 180,E1 20054.987,E2 20054.987} C_VEL
LIN {X 0,Y 409.932,Z 1253.866,A -85,B 0,C 180,E1 20052.248,E2 20052.248} C_VEL
LIN {X 0,Y 411.085,Z 1246.849,A -85,B 0,C 180,E1 20049.463,E2 20049.463} C_VEL
LIN {X 0,Y 412.71,Z 1238.72,A -85,B 0,C 180,E1 20046.668,E2 20046.668} C_VEL
LIN {X 0,Y 414.91,Z 1229.29,A -85,B 0,C 180,E1 20043.832,E2 20043.832} C_VEL
LIN {X 0,Y 418.058,Z 1217.128,A -85,B 0,C 180,E1 20040.64,E2 20040.64} C_VEL
LIN {X 0,Y 422.485,Z 1201.637,A -85,B 0,C 180,E1 20037.159,E2 20037.159} C_VEL
LIN {X 0,Y 426.664,Z 1187.905,A -85,B 0,C 180,E1 20034.466,E2 20034.466} C_VEL
LIN {X 0,Y 431.068,Z 1174.108,A -85,B 0,C 180,E1 20032.06,E2 20032.06} C_VEL
LIN {X 0,Y 436.414,Z 1157.712,A -85,B 0,C 180,E1 20029.523,E2 20029.523} C_VEL
LIN {X 0,Y 443.427,Z 1136.191,A -85,B 0,C 180,E1 20026.633,E2 20026.633} C_VEL
LIN {X 0,Y 449.155,Z 1118.543,A -85,B 0,C 180,E1 20024.573,E2 20024.573} C_VEL
LIN {X 0,Y 454.774,Z 1100.928,A -85,B 0,C 180,E1 20022.749,E2 20022.749} C_VEL
LIN {X 0,Y 461.406,Z 1079.436,A -85,B 0,C 180,E1 20020.793,E2 20020.793} C_VEL
LIN {X 0,Y 468.414,Z 1055.314,A -85,B 0,C 180,E1 20018.917,E2 20018.917} C_VEL
LIN {X 0,Y 474.092,Z 1034.66,A -85,B 0,C 180,E1 20017.534,E2 20017.534} C_VEL
LIN {X 0,Y 479.244,Z 1014.576,A -85,B 0,C 180,E1 20016.357,E2 20016.357} C_VEL
LIN {X 0,Y 484.931,Z 990.759,A -85,B 0,C 180,E1 20015.161,E2 20015.161} C_VEL
LIN {X 0,Y 490.736,Z 963.197,A -85,B 0,C 180,E1 20014.029,E2 20014.029} C_VEL
LIN {X 0,Y 494.94,Z 940.491,A -85,B 0,C 180,E1 20013.273,E2 20013.273} C_VEL
LIN {X 0,Y 498.593,Z 917.594,A -85,B 0,C 180,E1 20012.655,E2 20012.655} C_VEL
LIN {X 0,Y 502.113,Z 888.452,A -85,B 0,C 180,E1 20012.022,E2 20012.022} C_VEL
LIN {X 0,Y 507.203,Z 815.289,A -85,B 0,C 180,E1 20010.776,E2 20010.776} C_VEL
LIN {X 0,Y 521.563,Z 612.643,A -85,B 0,C 180,E1 20007.394,E2 20007.394} C_VEL
LIN {X 0,Y 527.864,Z 530.136,A -85,B 0,C 180,E1 20006.009,E2 20006.009} C_VEL
LIN {X 0,Y 517.222,Z 513.14,A -85,B 0,C 180,E1 20003.468,E2 20003.468} C_VEL
LIN {X 0,Y 506.883,Z 497.149,A -85,B 0,C 180,E1 20000.765,E2 20000.765} C_VEL
LIN {X 0,Y 497.389,Z 483.134,A -85,B 0,C 180,E1 19998.034,E2 19998.034} C_VEL
LIN {X 0,Y 489.386,Z 471.591,A -85,B 0,C 180,E1 19995.494,E2 19995.494} C_VEL
LIN {X 0,Y 480.345,Z 458.709,A -85,B 0,C 180,E1 19992.32,E2 19992.32} C_VEL
LIN {X 0,Y 472.368,Z 447.852,A -85,B 0,C 180,E1 19989.196,E2 19989.196} C_VEL
LIN {X 0,Y 467.13,Z 440.821,A -85,B 0,C 180,E1 19986.946,E2 19986.946} C_VEL
LIN {X 0,Y 464.206,Z 436.856,A -85,B 0,C 180,E1 19985.562,E2 19985.562} C_VEL
LIN {X 0,Y 460.015,Z 431.174,A -85,B 0,C 180,E1 19983.489,E2 19983.489} C_VEL
LIN {X 0,Y 455.819,Z 425.593,A -85,B 0,C 180,E1 19981.194,E2 19981.194} C_VEL
LIN {X 0,Y 451.723,Z 420.076,A -85,B 0,C 180,E1 19978.732,E2 19978.732} C_VEL
LIN {X 0,Y 447.473,Z 414.405,A -85,B 0,C 180,E1 19975.9,E2 19975.9} C_VEL
LIN {X 0,Y 444.443,Z 410.5,A -85,B 0,C 180,E1 19973.606,E2 19973.606} C_VEL
LIN {X 0,Y 443.251,Z 408.642,A -85,B 0,C 180,E1 19972.612,E2 19972.612} C_VEL
LIN {X 0,Y 440.219,Z 404.836,A -85,B 0,C 180,E1 19969.994,E2 19969.994} C_VEL
LIN {X 0,Y 439.139,Z 402.844,A -85,B 0,C 180,E1 19968.841,E2 19968.841} C_VEL
LIN {X 0,Y 436.142,Z 399.189,A -85,B 0,C 180,E1 19965.664,E2 19965.664} C_VEL
LIN {X 0,Y 435.066,Z 397.287,A -85,B 0,C 180,E1 19964.265,E2 19964.265} C_VEL
LIN {X 0,Y 431.924,Z 395.138,A -85,B 0,C 180,E1 19960.246,E2 19960.246} C_VEL
LIN {X 0,Y 430.15,Z 392.351,A -85,B 0,C 180,E1 19956.868,E2 19956.868} C_VEL
LIN {X 0,Y 429.478,Z 390.995,A -85,B 0,C 180,E1 19955.077,E2 19955.077} C_VEL
LIN {X 0,Y 427.941,Z 390.053,A -85,B 0,C 180,E1 19951.075,E2 19951.075} C_VEL
LIN {X 0,Y 427.054,Z 389.556,A -85,B 0,C 180,E1 19946.778,E2 19946.778} C_VEL
LIN {X 0,Y 427.01,Z 389.53,A -85,B 0,C 180,E1 19942.157,E2 19942.157} C_VEL
LIN {X 0,Y 427.751,Z 389.93,A -85,B 0,C 180,E1 19937.617,E2 19937.617} C_VEL
LIN {X 0,Y 429.374,Z 390.817,A -85,B 0,C 180,E1 19933.39,E2 19933.39} C_VEL
LIN {X 0,Y 430.324,Z 392.656,A -85,B 0,C 180,E1 19931.114,E2 19931.114} C_VEL
LIN {X 0,Y 432.638,Z 395.767,A -85,B 0,C 180,E1 19927.341,E2 19927.341} C_VEL
LIN {X 0,Y 435.964,Z 397.89,A -85,B 0,C 180,E1 19923.638,E2 19923.638} C_VEL
LIN {X 0,Y 437.765,Z 401.355,A -85,B 0,C 180,E1 19921.537,E2 19921.537} C_VEL
LIN {X 0,Y 440.899,Z 403.76,A -85,B 0,C 180,E1 19918.909,E2 19918.909} C_VEL
LIN {X 0,Y 441.974,Z 404.731,A -85,B 0,C 180,E1 19918.077,E2 19918.077} C_VEL
LIN {X 0,Y 444.13,Z 408.287,A -85,B 0,C 180,E1 19916.328,E2 19916.328} C_VEL
LIN {X 0,Y 447.672,Z 411.128,A -85,B 0,C 180,E1 19914.055,E2 19914.055} C_VEL
LIN {X 0,Y 450.013,Z 414.799,A -85,B 0,C 180,E1 19912.468,E2 19912.468} C_VEL
LIN {X 0,Y 453.34,Z 417.592,A -85,B 0,C 180,E1 19910.664,E2 19910.664} C_VEL
LIN {X 0,Y 456.322,Z 421.758,A -85,B 0,C 180,E1 19908.989,E2 19908.989} C_VEL
LIN {X 0,Y 458.776,Z 423.956,A -85,B 0,C 180,E1 19907.825,E2 19907.825} C_VEL
LIN {X 0,Y 462.09,Z 428.251,A -85,B 0,C 180,E1 19906.208,E2 19906.208} C_VEL
LIN {X 0,Y 464.108,Z 430.19,A -85,B 0,C 180,E1 19905.331,E2 19905.331} C_VEL
LIN {X 0,Y 468.122,Z 435.028,A -85,B 0,C 180,E1 19903.623,E2 19903.623} C_VEL
LIN {X 0,Y 469.929,Z 437.262,A -85,B 0,C 180,E1 19902.878,E2 19902.878} C_VEL
LIN {X 0,Y 474.749,Z 442.927,A -85,B 0,C 180,E1 19901.048,E2 19901.048} C_VEL
LIN {X 0,Y 479.766,Z 449.082,A -85,B 0,C 180,E1 19899.234,E2 19899.234} C_VEL
LIN {X 0,Y 484.732,Z 455.132,A -85,B 0,C 180,E1 19897.586,E2 19897.586} C_VEL
LIN {X 0,Y 492.285,Z 464.428,A -85,B 0,C 180,E1 19895.244,E2 19895.244} C_VEL
LIN {X 0,Y 504.495,Z 480.102,A -85,B 0,C 180,E1 19891.846,E2 19891.846} C_VEL
LIN {X 0,Y 516.373,Z 496.248,A -85,B 0,C 180,E1 19888.891,E2 19888.891} C_VEL
LIN {X 0,Y 523.783,Z 506.918,A -85,B 0,C 180,E1 19887.185,E2 19887.185} C_VEL
LIN {X 0,Y 508.783,Z 715.316,A -85,B 0,C 180,E1 19883.738,E2 19883.738} C_VEL
LIN {X 0,Y 504.166,Z 780.478,A -85,B 0,C 180,E1 19882.636,E2 19882.636} C_VEL
LIN {X 0,Y 501.059,Z 808.777,A -85,B 0,C 180,E1 19881.974,E2 19881.974} C_VEL
LIN {X 0,Y 497.862,Z 831.543,A -85,B 0,C 180,E1 19881.289,E2 19881.289} C_VEL
LIN {X 0,Y 494.313,Z 852.916,A -85,B 0,C 180,E1 19880.511,E2 19880.511} C_VEL
LIN {X 0,Y 494.121,Z 854.004,A -85,B 0,C 180,E1 19880.469,E2 19880.469} C_VEL
LIN {X 0,Y 492.186,Z 861.346,A -85,B 0,C 180,E1 19880.266,E2 19880.266} C_VEL
LIN {X 0,Y 484.655,Z 879.98,A -85,B 0,C 180,E1 19879.987,E2 19879.987} C_VEL
LIN {X 0,Y 482.445,Z 886.921,A -85,B 0,C 180,E1 19879.725,E2 19879.725} C_VEL
LIN {X 0,Y 477.429,Z 908.029,A -85,B 0,C 180,E1 19878.564,E2 19878.564} C_VEL
LIN {X 0,Y 471.301,Z 931.452,A -85,B 0,C 180,E1 19877.066,E2 19877.066} C_VEL
LIN {X 0,Y 464.615,Z 954.079,A -85,B 0,C 180,E1 19875.353,E2 19875.353} C_VEL
LIN {X 0,Y 458.731,Z 972.661,A -85,B 0,C 180,E1 19873.735,E2 19873.735} C_VEL
LIN {X 0,Y 453.328,Z 988.8,A -85,B 0,C 180,E1 19872.147,E2 19872.147} C_VEL
LIN {X 0,Y 447.295,Z 1005.975,A -85,B 0,C 180,E1 19870.24,E2 19870.24} C_VEL
LIN {X 0,Y 439.916,Z 1025.893,A -85,B 0,C 180,E1 19867.68,E2 19867.68} C_VEL
LIN {X 0,Y 433.714,Z 1041.918,A -85,B 0,C 180,E1 19865.277,E2 19865.277} C_VEL
LIN {X 0,Y 428.547,Z 1055.096,A -85,B 0,C 180,E1 19863.036,E2 19863.036} C_VEL
LIN {X 0,Y 423.654,Z 1067.497,A -85,B 0,C 180,E1 19860.655,E2 19860.655} C_VEL
LIN {X 0,Y 418.602,Z 1080.459,A -85,B 0,C 180,E1 19857.815,E2 19857.815} C_VEL
LIN {X 0,Y 413.471,Z 1093.836,A -85,B 0,C 180,E1 19854.346,E2 19854.346} C_VEL
LIN {X 0,Y 410.045,Z 1103.171,A -85,B 0,C 180,E1 19851.514,E2 19851.514} C_VEL
LIN {X 0,Y 407.298,Z 1111.224,A -85,B 0,C 180,E1 19848.696,E2 19848.696} C_VEL
LIN {X 0,Y 405.039,Z 1118.527,A -85,B 0,C 180,E1 19845.717,E2 19845.717} C_VEL
LIN {X 0,Y 403.243,Z 1125.033,A -85,B 0,C 180,E1 19842.571,E2 19842.571} C_VEL
LIN {X 0,Y 401.791,Z 1131.553,A -85,B 0,C 180,E1 19838.611,E2 19838.611} C_VEL
LIN {X 0,Y 401.132,Z 1135.596,A -85,B 0,C 180,E1 19835.331,E2 19835.331} C_VEL
LIN {X 0,Y 400.811,Z 1138.421,A -85,B 0,C 180,E1 19832.255,E2 19832.255} C_VEL
LIN {X 0,Y 400.682,Z 1140.203,A -85,B 0,C 180,E1 19829.436,E2 19829.436} C_VEL
LIN {X 0,Y 400.614,Z 1141.215,A -85,B 0,C 180,E1 19826.682,E2 19826.682} C_VEL
LIN {X 0,Y 400.663,Z 1141.491,A -85,B 0,C 180,E1 19823.847,E2 19823.847} C_VEL
LIN {X 0,Y 400.753,Z 1140.982,A -85,B 0,C 180,E1 19820.903,E2 19820.903} C_VEL
LIN {X 0,Y 400.955,Z 1139.688,A -85,B 0,C 180,E1 19818.013,E2 19818.013} C_VEL
LIN {X 0,Y 401.327,Z 1137.514,A -85,B 0,C 180,E1 19815.017,E2 19815.017} C_VEL
LIN {X 0,Y 402.055,Z 1134.187,A -85,B 0,C 180,E1 19811.767,E2 19811.767} C_VEL
LIN {X 0,Y 403.584,Z 1128.74,A -85,B 0,C 180,E1 19807.832,E2 19807.832} C_VEL
LIN {X 0,Y 405.681,Z 1122.486,A -85,B 0,C 180,E1 19804.382,E2 19804.382} C_VEL
LIN {X 0,Y 408.134,Z 1115.996,A -85,B 0,C 180,E1 19801.404,E2 19801.404} C_VEL
LIN {X 0,Y 411.923,Z 1106.976,A -85,B 0,C 180,E1 19797.913,E2 19797.913} C_VEL
LIN {X 0,Y 416.835,Z 1095.724,A -85,B 0,C 180,E1 19794.356,E2 19794.356} C_VEL
LIN {X 0,Y 421.353,Z 1085.812,A -85,B 0,C 180,E1 19791.677,E2 19791.677} C_VEL
LIN {X 0,Y 426.77,Z 1074.134,A -85,B 0,C 180,E1 19788.923,E2 19788.923} C_VEL
LIN {X 0,Y 433.806,Z 1058.828,A -85,B 0,C 180,E1 19785.858,E2 19785.858} C_VEL
LIN {X 0,Y 439.988,Z 1045.095,A -85,B 0,C 180,E1 19783.497,E2 19783.497} C_VEL
LIN {X 0,Y 447.458,Z 1028.164,A -85,B 0,C 180,E1 19780.958,E2 19780.958} C_VEL
LIN {X 0,Y 455.104,Z 1009.706,A -85,B 0,C 180,E1 19778.61,E2 19778.61} C_VEL
LIN {X 0,Y 462.098,Z 992.258,A -85,B 0,C 180,E1 19776.673,E2 19776.673} C_VEL
LIN {X 0,Y 470.395,Z 970.265,A -85,B 0,C 180,E1 19774.572,E2 19774.572} C_VEL
LIN {X 0,Y 478.878,Z 946.906,A -85,B 0,C 180,E1 19772.654,E2 19772.654} C_VEL
LIN {X 0,Y 488.902,Z 918.116,A -85,B 0,C 180,E1 19770.671,E2 19770.671} C_VEL
LIN {X 0,Y 499.496,Z 887.809,A -85,B 0,C 180,E1 19768.954,E2 19768.954} C_VEL
LIN {X 0,Y 500.859,Z 883.73,A -85,B 0,C 180,E1 19768.739,E2 19768.739} C_VEL
LIN {X 0,Y 488.08,Z 923.196,A -85,B 0,C 180,E1 19767.349,E2 19767.349} C_VEL
LIN {X 0,Y 477.81,Z 957.483,A -85,B 0,C 180,E1 19765.867,E2 19765.867} C_VEL
LIN {X 0,Y 468.127,Z 992.543,A -85,B 0,C 180,E1 19764.048,E2 19764.048} C_VEL
LIN {X 0,Y 460.44,Z 1021.382,A -85,B 0,C 180,E1 19762.295,E2 19762.295} C_VEL
LIN {X 0,Y 451.969,Z 1053.612,A -85,B 0,C 180,E1 19760.002,E2 19760.002} C_VEL
LIN {X 0,Y 445.884,Z 1076.458,A -85,B 0,C 180,E1 19758.116,E2 19758.116} C_VEL
LIN {X 0,Y 440.608,Z 1096.024,A -85,B 0,C 180,E1 19756.302,E2 19756.302} C_VEL
LIN {X 0,Y 435.486,Z 1114.766,A -85,B 0,C 180,E1 19754.361,E2 19754.361} C_VEL
LIN {X 0,Y 430.298,Z 1133.704,A -85,B 0,C 180,E1 19752.16,E2 19752.16} C_VEL
LIN {X 0,Y 424.128,Z 1156.111,A -85,B 0,C 180,E1 19749.183,E2 19749.183} C_VEL
LIN {X 0,Y 419.281,Z 1174.067,A -85,B 0,C 180,E1 19746.427,E2 19746.427} C_VEL
LIN {X 0,Y 415.067,Z 1190.001,A -85,B 0,C 180,E1 19743.646,E2 19743.646} C_VEL
LIN {X 0,Y 410.981,Z 1206.276,A -85,B 0,C 180,E1 19740.401,E2 19740.401} C_VEL
LIN {X 0,Y 407.573,Z 1220.866,A -85,B 0,C 180,E1 19736.991,E2 19736.991} C_VEL
LIN {X 0,Y 405.368,Z 1231.505,A -85,B 0,C 180,E1 19734.125,E2 19734.125} C_VEL
LIN {X 0,Y 403.72,Z 1240.545,A -85,B 0,C 180,E1 19731.35,E2 19731.35} C_VEL
LIN {X 0,Y 402.451,Z 1248.437,A -85,B 0,C 180,E1 19728.543,E2 19728.543} C_VEL
LIN {X 0,Y 401.654,Z 1254.869,A -85,B 0,C 180,E1 19725.892,E2 19725.892} C_VEL
LIN {X 0,Y 401.07,Z 1260.794,A -85,B 0,C 180,E1 19722.966,E2 19722.966} C_VEL
LIN {X 0,Y 400.785,Z 1265.296,A -85,B 0,C 180,E1 19720.203,E2 19720.203} C_VEL
LIN {X 0,Y 400.66,Z 1268.754,A -85,B 0,C 180,E1 19717.456,E2 19717.456} C_VEL
LIN {X 0,Y 400.651,Z 1271.187,A -85,B 0,C 180,E1 19714.724,E2 19714.724} C_VEL
LIN {X 0,Y 400.637,Z 1272.635,A -85,B 0,C 180,E1 19711.859,E2 19711.859} C_VEL
LIN {X 0,Y 400.575,Z 1272.981,A -85,B 0,C 180,E1 19709.142,E2 19709.142} C_VEL
LIN {X 0,Y 400.567,Z 1272.272,A -85,B 0,C 180,E1 19706.279,E2 19706.279} C_VEL
LIN {X 0,Y 400.532,Z 1270.46,A -85,B 0,C 180,E1 19703.406,E2 19703.406} C_VEL
LIN {X 0,Y 400.542,Z 1267.551,A -85,B 0,C 180,E1 19700.517,E2 19700.517} C_VEL
LIN {X 0,Y 400.798,Z 1263.56,A -85,B 0,C 180,E1 19697.611,E2 19697.611} C_VEL
LIN {X 0,Y 401.291,Z 1258.367,A -85,B 0,C 180,E1 19694.641,E2 19694.641} C_VEL
LIN {X 0,Y 402.094,Z 1252.336,A -85,B 0,C 180,E1 19691.792,E2 19691.792} C_VEL
LIN {X 0,Y 403.358,Z 1245.23,A -85,B 0,C 180,E1 19688.934,E2 19688.934} C_VEL
LIN {X 0,Y 405.055,Z 1237.13,A -85,B 0,C 180,E1 19686.119,E2 19686.119} C_VEL
LIN {X 0,Y 407.424,Z 1227.357,A -85,B 0,C 180,E1 19683.156,E2 19683.156} C_VEL
LIN {X 0,Y 411.157,Z 1213.91,A -85,B 0,C 180,E1 19679.614,E2 19679.614} C_VEL
LIN {X 0,Y 415.464,Z 1199.469,A -85,B 0,C 180,E1 19676.379,E2 19676.379} C_VEL
LIN {X 0,Y 419.673,Z 1186.306,A -85,B 0,C 180,E1 19673.782,E2 19673.782} C_VEL
LIN {X 0,Y 424.49,Z 1171.76,A -85,B 0,C 180,E1 19671.231,E2 19671.231} C_VEL
LIN {X 0,Y 430.786,Z 1153.242,A -85,B 0,C 180,E1 19668.365,E2 19668.365} C_VEL
LIN {X 0,Y 437.498,Z 1133.251,A -85,B 0,C 180,E1 19665.717,E2 19665.717} C_VEL
LIN {X 0,Y 443.209,Z 1116.156,A -85,B 0,C 180,E1 19663.729,E2 19663.729} C_VEL
LIN {X 0,Y 449.548,Z 1096.781,A -85,B 0,C 180,E1 19661.737,E2 19661.737} C_VEL
LIN {X 0,Y 457.482,Z 1071.531,A -85,B 0,C 180,E1 19659.51,E2 19659.51} C_VEL
LIN {X 0,Y 463.56,Z 1051.024,A -85,B 0,C 180,E1 19657.957,E2 19657.957} C_VEL
LIN {X 0,Y 469.41,Z 1030.153,A -85,B 0,C 180,E1 19656.579,E2 19656.579} C_VEL
LIN {X 0,Y 476.105,Z 1004.406,A -85,B 0,C 180,E1 19655.131,E2 19655.131} C_VEL
LIN {X 0,Y 481.925,Z 979.133,A -85,B 0,C 180,E1 19653.965,E2 19653.965} C_VEL
LIN {X 0,Y 486.647,Z 956.483,A -85,B 0,C 180,E1 19653.095,E2 19653.095} C_VEL
LIN {X 0,Y 491.605,Z 929.411,A -85,B 0,C 180,E1 19652.247,E2 19652.247} C_VEL
LIN {X 0,Y 495.573,Z 901.61,A -85,B 0,C 180,E1 19651.584,E2 19651.584} C_VEL
LIN {X 0,Y 497.985,Z 877.384,A -85,B 0,C 180,E1 19651.105,E2 19651.105} C_VEL
LIN {X 0,Y 513.305,Z 664.317,A -85,B 0,C 180,E1 19647.516,E2 19647.516} C_VEL
LIN {X 0,Y 523.321,Z 534.331,A -85,B 0,C 180,E1 19645.31,E2 19645.31} C_VEL
LIN {X 0,Y 511.38,Z 515.123,A -85,B 0,C 180,E1 19642.352,E2 19642.352} C_VEL
LIN {X 0,Y 500.467,Z 498.496,A -85,B 0,C 180,E1 19639.369,E2 19639.369} C_VEL
LIN {X 0,Y 491.005,Z 484.462,A -85,B 0,C 180,E1 19636.504,E2 19636.504} C_VEL
LIN {X 0,Y 481.51,Z 470.879,A -85,B 0,C 180,E1 19633.296,E2 19633.296} C_VEL
LIN {X 0,Y 473.659,Z 459.957,A -85,B 0,C 180,E1 19630.337,E2 19630.337} C_VEL
LIN {X 0,Y 469.536,Z 454.376,A -85,B 0,C 180,E1 19628.635,E2 19628.635} C_VEL
LIN {X 0,Y 465.469,Z 448.735,A -85,B 0,C 180,E1 19626.847,E2 19626.847} C_VEL
LIN {X 0,Y 462.14,Z 444.252,A -85,B 0,C 180,E1 19625.276,E2 19625.276} C_VEL
LIN {X 0,Y 457.987,Z 438.581,A -85,B 0,C 180,E1 19623.191,E2 19623.191} C_VEL
